DATA_BLOCK "ManualOperationControl_U1Em6"   // DB199
// stored: MemoryReserve 100
   VAR
      manualOperationEm { ExternalAccessible := 'False'; ExternalVisible := 'False'; ExternalWritable := 'False'} : "LAF_typeManEm";
      manualOperationEmArea { ExternalAccessible := 'False'; ExternalVisible := 'False'; ExternalWritable := 'False'} : Array[1..2] of "LAF_typeManOperationArea";
      manualOperationCms { ExternalAccessible := 'False'; ExternalVisible := 'False'; ExternalWritable := 'False'} : Array[1..90] of "LAF_typeManOperation";
      axis { ExternalAccessible := 'False'; ExternalVisible := 'False'; ExternalWritable := 'False'} : Array[0..0] of "LBC_typeAxisControlInterface";
      axis64Pos { S7_SetPoint := 'True'} : Array[0..20] of "LBC_typeAxis64PosInterface";
      softCam { S7_SetPoint := 'True'} : Array[0..20] of "LER_typeSoftCamInterface2";
      twoWayActuator { S7_SetPoint := 'True'} : Array[0..14] of "LBC_typeTwoWayActuatorInterface";
   END_VAR
BEGIN
   manualOperationEm.equipmentModuleNum := 1070;
   manualOperationEm.actvArea := 0;
   manualOperationEm.pages.total := 0;
   manualOperationEm.pages.actv := 0;
   manualOperationEm.pages.numOfActvItems := 0;
   manualOperationEmArea[1..2].areaNum := 0;
   manualOperationEmArea[1].displayedLines := '6-18;';
   manualOperationEmArea[2].displayedLines := '21-26;';
   manualOperationEmArea[1..2].hmiPage.total := 0;
   manualOperationEmArea[1..2].hmiPage.actv := 0;
   manualOperationEmArea[1..2].hmiPage.numOfActvItems := 0;
   manualOperationCms[1..90].intf.lineNum := 0;
   manualOperationCms[1..90].intf.mode := 1;
   manualOperationCms[1..90].intf.showLine := FALSE;
   manualOperationCms[1..90].intf.enableMechAddr := FALSE;
   manualOperationCms[1..90].intf.expandable := FALSE;
   manualOperationCms[1..90].intf.disableLineSel := FALSE;
   manualOperationCms[1..90].intf.enableBigArea := FALSE;
   manualOperationCms[1..90].intf.cnfrmExecLeft := FALSE;
   manualOperationCms[1..90].intf.cnfrmExecRight := FALSE;
   manualOperationCms[1..90].intf.disableLeft := FALSE;
   manualOperationCms[1..90].intf.disableRight := FALSE;
   manualOperationCms[1..90].intf.cnfrmExecLeftCmd := FALSE;
   manualOperationCms[1..90].intf.cnfrmExecRightCmd := FALSE;
   manualOperationCms[1..90].intf.fieldDevAckLeft := FALSE;
   manualOperationCms[1..90].intf.fieldDevAckRight := FALSE;
   manualOperationCms[1..90].intf.nextLeftEndPos := 0;
   manualOperationCms[1..90].intf.nextRightEndPos := 0;
   manualOperationCms[1].intf.leftEndPosSens[0..7] := FALSE;
   manualOperationCms[2].intf.leftEndPosSens[0..7] := FALSE;
   manualOperationCms[3].intf.leftEndPosSens[0..7] := FALSE;
   manualOperationCms[4].intf.leftEndPosSens[0..7] := FALSE;
   manualOperationCms[5].intf.leftEndPosSens[0..7] := FALSE;
   manualOperationCms[6].intf.leftEndPosSens[0..7] := FALSE;
   manualOperationCms[7].intf.leftEndPosSens[0..7] := FALSE;
   manualOperationCms[8].intf.leftEndPosSens[0..7] := FALSE;
   manualOperationCms[9].intf.leftEndPosSens[0..7] := FALSE;
   manualOperationCms[10].intf.leftEndPosSens[0..7] := FALSE;
   manualOperationCms[11].intf.leftEndPosSens[0..7] := FALSE;
   manualOperationCms[12].intf.leftEndPosSens[0..7] := FALSE;
   manualOperationCms[13].intf.leftEndPosSens[0..7] := FALSE;
   manualOperationCms[14].intf.leftEndPosSens[0..7] := FALSE;
   manualOperationCms[15].intf.leftEndPosSens[0..7] := FALSE;
   manualOperationCms[16].intf.leftEndPosSens[0..7] := FALSE;
   manualOperationCms[17].intf.leftEndPosSens[0..7] := FALSE;
   manualOperationCms[18].intf.leftEndPosSens[0..7] := FALSE;
   manualOperationCms[19].intf.leftEndPosSens[0..7] := FALSE;
   manualOperationCms[20].intf.leftEndPosSens[0..7] := FALSE;
   manualOperationCms[21].intf.leftEndPosSens[0..7] := FALSE;
   manualOperationCms[22].intf.leftEndPosSens[0..7] := FALSE;
   manualOperationCms[23].intf.leftEndPosSens[0..7] := FALSE;
   manualOperationCms[24].intf.leftEndPosSens[0..7] := FALSE;
   manualOperationCms[25].intf.leftEndPosSens[0..7] := FALSE;
   manualOperationCms[26].intf.leftEndPosSens[0..7] := FALSE;
   manualOperationCms[27].intf.leftEndPosSens[0..7] := FALSE;
   manualOperationCms[28].intf.leftEndPosSens[0..7] := FALSE;
   manualOperationCms[29].intf.leftEndPosSens[0..7] := FALSE;
   manualOperationCms[30].intf.leftEndPosSens[0..7] := FALSE;
   manualOperationCms[31].intf.leftEndPosSens[0..7] := FALSE;
   manualOperationCms[32].intf.leftEndPosSens[0..7] := FALSE;
   manualOperationCms[33].intf.leftEndPosSens[0..7] := FALSE;
   manualOperationCms[34].intf.leftEndPosSens[0..7] := FALSE;
   manualOperationCms[35].intf.leftEndPosSens[0..7] := FALSE;
   manualOperationCms[36].intf.leftEndPosSens[0..7] := FALSE;
   manualOperationCms[37].intf.leftEndPosSens[0..7] := FALSE;
   manualOperationCms[38].intf.leftEndPosSens[0..7] := FALSE;
   manualOperationCms[39].intf.leftEndPosSens[0..7] := FALSE;
   manualOperationCms[40].intf.leftEndPosSens[0..7] := FALSE;
   manualOperationCms[41].intf.leftEndPosSens[0..7] := FALSE;
   manualOperationCms[42].intf.leftEndPosSens[0..7] := FALSE;
   manualOperationCms[43].intf.leftEndPosSens[0..7] := FALSE;
   manualOperationCms[44].intf.leftEndPosSens[0..7] := FALSE;
   manualOperationCms[45].intf.leftEndPosSens[0..7] := FALSE;
   manualOperationCms[46].intf.leftEndPosSens[0..7] := FALSE;
   manualOperationCms[47].intf.leftEndPosSens[0..7] := FALSE;
   manualOperationCms[48].intf.leftEndPosSens[0..7] := FALSE;
   manualOperationCms[49].intf.leftEndPosSens[0..7] := FALSE;
   manualOperationCms[50].intf.leftEndPosSens[0..7] := FALSE;
   manualOperationCms[51].intf.leftEndPosSens[0..7] := FALSE;
   manualOperationCms[52].intf.leftEndPosSens[0..7] := FALSE;
   manualOperationCms[53].intf.leftEndPosSens[0..7] := FALSE;
   manualOperationCms[54].intf.leftEndPosSens[0..7] := FALSE;
   manualOperationCms[55].intf.leftEndPosSens[0..7] := FALSE;
   manualOperationCms[56].intf.leftEndPosSens[0..7] := FALSE;
   manualOperationCms[57].intf.leftEndPosSens[0..7] := FALSE;
   manualOperationCms[58].intf.leftEndPosSens[0..7] := FALSE;
   manualOperationCms[59].intf.leftEndPosSens[0..7] := FALSE;
   manualOperationCms[60].intf.leftEndPosSens[0..7] := FALSE;
   manualOperationCms[61].intf.leftEndPosSens[0..7] := FALSE;
   manualOperationCms[62].intf.leftEndPosSens[0..7] := FALSE;
   manualOperationCms[63].intf.leftEndPosSens[0..7] := FALSE;
   manualOperationCms[64].intf.leftEndPosSens[0..7] := FALSE;
   manualOperationCms[65].intf.leftEndPosSens[0..7] := FALSE;
   manualOperationCms[66].intf.leftEndPosSens[0..7] := FALSE;
   manualOperationCms[67].intf.leftEndPosSens[0..7] := FALSE;
   manualOperationCms[68].intf.leftEndPosSens[0..7] := FALSE;
   manualOperationCms[69].intf.leftEndPosSens[0..7] := FALSE;
   manualOperationCms[70].intf.leftEndPosSens[0..7] := FALSE;
   manualOperationCms[71].intf.leftEndPosSens[0..7] := FALSE;
   manualOperationCms[72].intf.leftEndPosSens[0..7] := FALSE;
   manualOperationCms[73].intf.leftEndPosSens[0..7] := FALSE;
   manualOperationCms[74].intf.leftEndPosSens[0..7] := FALSE;
   manualOperationCms[75].intf.leftEndPosSens[0..7] := FALSE;
   manualOperationCms[76].intf.leftEndPosSens[0..7] := FALSE;
   manualOperationCms[77].intf.leftEndPosSens[0..7] := FALSE;
   manualOperationCms[78].intf.leftEndPosSens[0..7] := FALSE;
   manualOperationCms[79].intf.leftEndPosSens[0..7] := FALSE;
   manualOperationCms[80].intf.leftEndPosSens[0..7] := FALSE;
   manualOperationCms[81].intf.leftEndPosSens[0..7] := FALSE;
   manualOperationCms[82].intf.leftEndPosSens[0..7] := FALSE;
   manualOperationCms[83].intf.leftEndPosSens[0..7] := FALSE;
   manualOperationCms[84].intf.leftEndPosSens[0..7] := FALSE;
   manualOperationCms[85].intf.leftEndPosSens[0..7] := FALSE;
   manualOperationCms[86].intf.leftEndPosSens[0..7] := FALSE;
   manualOperationCms[87].intf.leftEndPosSens[0..7] := FALSE;
   manualOperationCms[88].intf.leftEndPosSens[0..7] := FALSE;
   manualOperationCms[89].intf.leftEndPosSens[0..7] := FALSE;
   manualOperationCms[90].intf.leftEndPosSens[0..7] := FALSE;
   manualOperationCms[1].intf.rightEndPosSens[0..7] := FALSE;
   manualOperationCms[2].intf.rightEndPosSens[0..7] := FALSE;
   manualOperationCms[3].intf.rightEndPosSens[0..7] := FALSE;
   manualOperationCms[4].intf.rightEndPosSens[0..7] := FALSE;
   manualOperationCms[5].intf.rightEndPosSens[0..7] := FALSE;
   manualOperationCms[6].intf.rightEndPosSens[0..7] := FALSE;
   manualOperationCms[7].intf.rightEndPosSens[0..7] := FALSE;
   manualOperationCms[8].intf.rightEndPosSens[0..7] := FALSE;
   manualOperationCms[9].intf.rightEndPosSens[0..7] := FALSE;
   manualOperationCms[10].intf.rightEndPosSens[0..7] := FALSE;
   manualOperationCms[11].intf.rightEndPosSens[0..7] := FALSE;
   manualOperationCms[12].intf.rightEndPosSens[0..7] := FALSE;
   manualOperationCms[13].intf.rightEndPosSens[0..7] := FALSE;
   manualOperationCms[14].intf.rightEndPosSens[0..7] := FALSE;
   manualOperationCms[15].intf.rightEndPosSens[0..7] := FALSE;
   manualOperationCms[16].intf.rightEndPosSens[0..7] := FALSE;
   manualOperationCms[17].intf.rightEndPosSens[0..7] := FALSE;
   manualOperationCms[18].intf.rightEndPosSens[0..7] := FALSE;
   manualOperationCms[19].intf.rightEndPosSens[0..7] := FALSE;
   manualOperationCms[20].intf.rightEndPosSens[0..7] := FALSE;
   manualOperationCms[21].intf.rightEndPosSens[0..7] := FALSE;
   manualOperationCms[22].intf.rightEndPosSens[0..7] := FALSE;
   manualOperationCms[23].intf.rightEndPosSens[0..7] := FALSE;
   manualOperationCms[24].intf.rightEndPosSens[0..7] := FALSE;
   manualOperationCms[25].intf.rightEndPosSens[0..7] := FALSE;
   manualOperationCms[26].intf.rightEndPosSens[0..7] := FALSE;
   manualOperationCms[27].intf.rightEndPosSens[0..7] := FALSE;
   manualOperationCms[28].intf.rightEndPosSens[0..7] := FALSE;
   manualOperationCms[29].intf.rightEndPosSens[0..7] := FALSE;
   manualOperationCms[30].intf.rightEndPosSens[0..7] := FALSE;
   manualOperationCms[31].intf.rightEndPosSens[0..7] := FALSE;
   manualOperationCms[32].intf.rightEndPosSens[0..7] := FALSE;
   manualOperationCms[33].intf.rightEndPosSens[0..7] := FALSE;
   manualOperationCms[34].intf.rightEndPosSens[0..7] := FALSE;
   manualOperationCms[35].intf.rightEndPosSens[0..7] := FALSE;
   manualOperationCms[36].intf.rightEndPosSens[0..7] := FALSE;
   manualOperationCms[37].intf.rightEndPosSens[0..7] := FALSE;
   manualOperationCms[38].intf.rightEndPosSens[0..7] := FALSE;
   manualOperationCms[39].intf.rightEndPosSens[0..7] := FALSE;
   manualOperationCms[40].intf.rightEndPosSens[0..7] := FALSE;
   manualOperationCms[41].intf.rightEndPosSens[0..7] := FALSE;
   manualOperationCms[42].intf.rightEndPosSens[0..7] := FALSE;
   manualOperationCms[43].intf.rightEndPosSens[0..7] := FALSE;
   manualOperationCms[44].intf.rightEndPosSens[0..7] := FALSE;
   manualOperationCms[45].intf.rightEndPosSens[0..7] := FALSE;
   manualOperationCms[46].intf.rightEndPosSens[0..7] := FALSE;
   manualOperationCms[47].intf.rightEndPosSens[0..7] := FALSE;
   manualOperationCms[48].intf.rightEndPosSens[0..7] := FALSE;
   manualOperationCms[49].intf.rightEndPosSens[0..7] := FALSE;
   manualOperationCms[50].intf.rightEndPosSens[0..7] := FALSE;
   manualOperationCms[51].intf.rightEndPosSens[0..7] := FALSE;
   manualOperationCms[52].intf.rightEndPosSens[0..7] := FALSE;
   manualOperationCms[53].intf.rightEndPosSens[0..7] := FALSE;
   manualOperationCms[54].intf.rightEndPosSens[0..7] := FALSE;
   manualOperationCms[55].intf.rightEndPosSens[0..7] := FALSE;
   manualOperationCms[56].intf.rightEndPosSens[0..7] := FALSE;
   manualOperationCms[57].intf.rightEndPosSens[0..7] := FALSE;
   manualOperationCms[58].intf.rightEndPosSens[0..7] := FALSE;
   manualOperationCms[59].intf.rightEndPosSens[0..7] := FALSE;
   manualOperationCms[60].intf.rightEndPosSens[0..7] := FALSE;
   manualOperationCms[61].intf.rightEndPosSens[0..7] := FALSE;
   manualOperationCms[62].intf.rightEndPosSens[0..7] := FALSE;
   manualOperationCms[63].intf.rightEndPosSens[0..7] := FALSE;
   manualOperationCms[64].intf.rightEndPosSens[0..7] := FALSE;
   manualOperationCms[65].intf.rightEndPosSens[0..7] := FALSE;
   manualOperationCms[66].intf.rightEndPosSens[0..7] := FALSE;
   manualOperationCms[67].intf.rightEndPosSens[0..7] := FALSE;
   manualOperationCms[68].intf.rightEndPosSens[0..7] := FALSE;
   manualOperationCms[69].intf.rightEndPosSens[0..7] := FALSE;
   manualOperationCms[70].intf.rightEndPosSens[0..7] := FALSE;
   manualOperationCms[71].intf.rightEndPosSens[0..7] := FALSE;
   manualOperationCms[72].intf.rightEndPosSens[0..7] := FALSE;
   manualOperationCms[73].intf.rightEndPosSens[0..7] := FALSE;
   manualOperationCms[74].intf.rightEndPosSens[0..7] := FALSE;
   manualOperationCms[75].intf.rightEndPosSens[0..7] := FALSE;
   manualOperationCms[76].intf.rightEndPosSens[0..7] := FALSE;
   manualOperationCms[77].intf.rightEndPosSens[0..7] := FALSE;
   manualOperationCms[78].intf.rightEndPosSens[0..7] := FALSE;
   manualOperationCms[79].intf.rightEndPosSens[0..7] := FALSE;
   manualOperationCms[80].intf.rightEndPosSens[0..7] := FALSE;
   manualOperationCms[81].intf.rightEndPosSens[0..7] := FALSE;
   manualOperationCms[82].intf.rightEndPosSens[0..7] := FALSE;
   manualOperationCms[83].intf.rightEndPosSens[0..7] := FALSE;
   manualOperationCms[84].intf.rightEndPosSens[0..7] := FALSE;
   manualOperationCms[85].intf.rightEndPosSens[0..7] := FALSE;
   manualOperationCms[86].intf.rightEndPosSens[0..7] := FALSE;
   manualOperationCms[87].intf.rightEndPosSens[0..7] := FALSE;
   manualOperationCms[88].intf.rightEndPosSens[0..7] := FALSE;
   manualOperationCms[89].intf.rightEndPosSens[0..7] := FALSE;
   manualOperationCms[90].intf.rightEndPosSens[0..7] := FALSE;
   manualOperationCms[1..90].intf.pos := 0.0;
   manualOperationCms[1..90].intf.minPos := 0.0;
   manualOperationCms[1..90].intf.maxPos := 0.0;
   manualOperationCms[1..90].intf.showPos := 0;
   manualOperationCms[1..90].cmd.lineSel := FALSE;
   manualOperationCms[1..90].cmd.expandedOemArea := FALSE;
   manualOperationCms[1..90].cmd.execLeftCmd := FALSE;
   manualOperationCms[1..90].cmd.execRightCmd := FALSE;
   manualOperationCms[1..90].cmd.disableLeftClick := FALSE;
   manualOperationCms[1..90].cmd.disableRightClick := FALSE;
   manualOperationCms[1..90].cmd.moreInfo := FALSE;
   manualOperationCms[1..90].cmd.actvAddr := 1;
   axis[0].commandConfiguration.generalSettings.stopOnError := TRUE;
   axis[0].commandConfiguration.generalSettings.resetWithRestart := FALSE;
   axis[0].commandConfiguration.generalSettings.abortWaitingSyncCmd := TRUE;
   axis[0].commandConfiguration.power.startMode := 1;
   axis[0].commandConfiguration.power.stopMode := 0;
   axis[0].commandConfiguration.power.syncMotionSimulation := FALSE;
   axis[0].commandConfiguration.power.syncMotionSimulationExtendedMode := -1;
   axis[0].commandConfiguration.jog.velocity := 0.0;
   axis[0].commandConfiguration.jog.acceleration := -1.0;
   axis[0].commandConfiguration.jog.deceleration := -1.0;
   axis[0].commandConfiguration.jog.jerk := -1.0;
   axis[0].commandConfiguration.jog.positionControlled := TRUE;
   axis[0].commandConfiguration.jog.increment := 0.0;
   axis[0].commandConfiguration.jog.mode := 0;
   axis[0].commandConfiguration.moveVelocity.velocity := 0.0;
   axis[0].commandConfiguration.moveVelocity.acceleration := -1.0;
   axis[0].commandConfiguration.moveVelocity.deceleration := -1.0;
   axis[0].commandConfiguration.moveVelocity.jerk := -1.0;
   axis[0].commandConfiguration.moveVelocity.direction := 0;
   axis[0].commandConfiguration.moveVelocity.positionControlled := TRUE;
   axis[0].commandConfiguration.moveVelocity.velocityChangeOnTheFly := FALSE;
   axis[0].commandConfiguration.stop.deceleration := -1.0;
   axis[0].commandConfiguration.stop.jerk := -1.0;
   axis[0].commandConfiguration.stop.abortAcceleration := FALSE;
   axis[0].commandConfiguration.fastStop.deceleration := -1.0;
   axis[0].commandConfiguration.fastStop.jerk := -1.0;
   axis[0].commandConfiguration.fastStop.abortAcceleration := FALSE;
   axis[0].commandConfiguration.fastStop.replaceStopPossible := FALSE;
   axis[0].commandConfiguration.torqueLimiting.limit := -1.0;
   axis[0].commandConfiguration.torqueLimiting.mode := 0;
   axis[0].commandConfiguration.homing.position := 0.0;
   axis[0].commandConfiguration.homing.mode := 0;
   axis[0].commandConfiguration.homing.sensor := 0;
   axis[0].commandConfiguration.homing.extendedMode := -1;
   axis[0].commandConfiguration.homing.extendedModeTorqueLimit := 0.0;
   axis[0].commandConfiguration.homing.extendedModeTargetPosition := 0.0;
   axis[0].commandConfiguration.posRelative.distance := 0.0;
   axis[0].commandConfiguration.posRelative.velocity := -1.0;
   axis[0].commandConfiguration.posRelative.acceleration := -1.0;
   axis[0].commandConfiguration.posRelative.deceleration := -1.0;
   axis[0].commandConfiguration.posRelative.jerk := -1.0;
   axis[0].commandConfiguration.posRelative.direction := 0;
   axis[0].commandConfiguration.posAbsolute.position := 0.0;
   axis[0].commandConfiguration.posAbsolute.velocity := -1.0;
   axis[0].commandConfiguration.posAbsolute.acceleration := -1.0;
   axis[0].commandConfiguration.posAbsolute.deceleration := -1.0;
   axis[0].commandConfiguration.posAbsolute.jerk := -1.0;
   axis[0].commandConfiguration.posAbsolute.direction := 1;
   axis[0].commandConfiguration.posAbsolute.positionChangeOnTheFly := FALSE;
   axis[0].commandConfiguration.posAbsolute.velocityChangeOnTheFly := FALSE;
   axis[0].commandConfiguration.posSuperimposed.distance := 0.0;
   axis[0].commandConfiguration.posSuperimposed.velocityDiff := -1.0;
   axis[0].commandConfiguration.posSuperimposed.acceleration := -1.0;
   axis[0].commandConfiguration.posSuperimposed.deceleration := -1.0;
   axis[0].commandConfiguration.posSuperimposed.jerk := -1.0;
   axis[0].commandConfiguration.posSuperimposed.direction := 0;
   axis[0].commandConfiguration.haltSuperimposed.deceleration := -1.0;
   axis[0].commandConfiguration.haltSuperimposed.jerk := -1.0;
   axis[0].commandConfiguration.haltSuperimposed.abortAcceleration := FALSE;
   axis[0].commandConfiguration.gearInRelative.ratioNumerator := 1;
   axis[0].commandConfiguration.gearInRelative.ratioDenominator := 1;
   axis[0].commandConfiguration.gearInRelative.acceleration := -1.0;
   axis[0].commandConfiguration.gearInRelative.deceleration := -1.0;
   axis[0].commandConfiguration.gearInRelative.jerk := -1.0;
   axis[0].commandConfiguration.gearInRelative.ratioChangeOnTheFly := FALSE;
   axis[0].commandConfiguration.gearInAbsolute.ratioNumerator := 1;
   axis[0].commandConfiguration.gearInAbsolute.ratioDenominator := 1;
   axis[0].commandConfiguration.gearInAbsolute.masterSyncPosition := 0.0;
   axis[0].commandConfiguration.gearInAbsolute.slaveSyncPosition := 0.0;
   axis[0].commandConfiguration.gearInAbsolute.syncProfileReference := 1;
   axis[0].commandConfiguration.gearInAbsolute.masterStartDistance := 0.0;
   axis[0].commandConfiguration.gearInAbsolute.velocity := -1.0;
   axis[0].commandConfiguration.gearInAbsolute.acceleration := -1.0;
   axis[0].commandConfiguration.gearInAbsolute.deceleration := -1.0;
   axis[0].commandConfiguration.gearInAbsolute.jerk := -1.0;
   axis[0].commandConfiguration.gearInAbsolute.syncDirection := 1;
   axis[0].commandConfiguration.gearInAbsolute.ratioChangeOnTheFly := FALSE;
   axis[0].commandConfiguration.gearInVelocity.continuousUpdate := FALSE;
   axis[0].commandConfiguration.gearInVelocity.ratioNumerator := 1;
   axis[0].commandConfiguration.gearInVelocity.ratioDenominator := 1;
   axis[0].commandConfiguration.gearInVelocity.acceleration := -1.0;
   axis[0].commandConfiguration.gearInVelocity.deceleration := -1.0;
   axis[0].commandConfiguration.gearInVelocity.jerk := -1.0;
   axis[0].commandConfiguration.gearInVelocity.positionControlled := FALSE;
   axis[0].commandConfiguration.camIn.masterOffset := 0.0;
   axis[0].commandConfiguration.camIn.slaveOffset := 0.0;
   axis[0].commandConfiguration.camIn.masterScaling := 1.0;
   axis[0].commandConfiguration.camIn.slaveScaling := 1.0;
   axis[0].commandConfiguration.camIn.masterSyncPosition := 0.0;
   axis[0].commandConfiguration.camIn.syncProfileReference := 1;
   axis[0].commandConfiguration.camIn.masterStartDistance := 0.0;
   axis[0].commandConfiguration.camIn.velocity := -1.0;
   axis[0].commandConfiguration.camIn.acceleration := -1.0;
   axis[0].commandConfiguration.camIn.deceleration := -1.0;
   axis[0].commandConfiguration.camIn.jerk := -1.0;
   axis[0].commandConfiguration.camIn.applicationMode := 0;
   axis[0].commandConfiguration.camIn.syncDirection := 1;
   axis[0].commandConfiguration.gearOutCamOut.slavePosition := 0.0;
   axis[0].commandConfiguration.gearOutCamOut.syncProfileReference := 1;
   axis[0].commandConfiguration.gearOutCamOut.masterStopDistance := 0.0;
   axis[0].commandConfiguration.gearOutCamOut.deceleration := -1.0;
   axis[0].commandConfiguration.gearOutCamOut.jerk := -1.0;
   axis[0].commandConfiguration.gearOutCamOut.syncOutDirection := 3;
   axis[0].commandConfiguration.gearOutCamOut.gearOutCamOutMode := -1;
   axis[0].commandConfiguration.phasing.phaseShift := 0.0;
   axis[0].commandConfiguration.phasing.velocity := -1.0;
   axis[0].commandConfiguration.phasing.acceleration := -1.0;
   axis[0].commandConfiguration.phasing.deceleration := -1.0;
   axis[0].commandConfiguration.phasing.jerk := -1.0;
   axis[0].commandConfiguration.phasing.profileReference := 0;
   axis[0].commandConfiguration.phasing.phasingDistance := 0.0;
   axis[0].commandConfiguration.phasing.startPosition := 0.0;
   axis[0].commandConfiguration.phasing.direction := 3;
   axis[0].commandConfiguration.phasing.phaseAbsolute := TRUE;
   axis[0].commandConfiguration.phasing.phaseShiftChangeOnTheFly := FALSE;
   axis[0].commandConfiguration.offset.offset := 0.0;
   axis[0].commandConfiguration.offset.profileReference := 1;
   axis[0].commandConfiguration.offset.offsetDistance := 0.0;
   axis[0].commandConfiguration.offset.startPosition := 0.0;
   axis[0].commandConfiguration.offset.direction := 3;
   axis[0].commandConfiguration.offset.offsetAbsolute := TRUE;
   axis[0].commandConfiguration.offset.offsetChangeOnTheFly := FALSE;
   axis[0].commands.enable := FALSE;
   axis[0].commands.enableAxis := FALSE;
   axis[0].commands.resetAxis := FALSE;
   axis[0].commands.openBrake := FALSE;
   axis[0].commands.jogForward := FALSE;
   axis[0].commands.jogBackward := FALSE;
   axis[0].commands.moveVelocity := FALSE;
   axis[0].commands.stop := FALSE;
   axis[0].commands.fastStop := FALSE;
   axis[0].commands.torqueLimiting := FALSE;
   axis[0].commands.homing := FALSE;
   axis[0].commands.posRelative := FALSE;
   axis[0].commands.posAbsolute := FALSE;
   axis[0].commands.posSuperimposed := FALSE;
   axis[0].commands.haltSuperimposed := FALSE;
   axis[0].commands.gearInRelative := FALSE;
   axis[0].commands.gearInAbsolute := FALSE;
   axis[0].commands.gearInVelocity := FALSE;
   axis[0].commands.camIn := FALSE;
   axis[0].commands.gearOutCamOut := FALSE;
   axis[0].commands.phasing := FALSE;
   axis[0].commands.offset := FALSE;
   axis[0].commands.refreshConfiguration := FALSE;
   axis[0].commands.editConfiguration := FALSE;
   axis[0].commands.saveConfiguration := FALSE;
   axis[0].commands.uploadCurrentTorque := FALSE;
   axis[0].commands.reset := FALSE;
   axis[0].monitoring.enable := FALSE;
   axis[0].monitoring.referenceDesignator := WSTRING#'';
   axis[0].monitoring.enabled := FALSE;
   axis[0].monitoring.resetAxis := FALSE;
   axis[0].monitoring.moveVelocity := FALSE;
   axis[0].monitoring.fastStop := FALSE;
   axis[0].monitoring.stop := FALSE;
   axis[0].monitoring.homing := FALSE;
   axis[0].monitoring.posRelative := FALSE;
   axis[0].monitoring.posAbsolute := FALSE;
   axis[0].monitoring.posSuperimposed := FALSE;
   axis[0].monitoring.haltSuperimposed := FALSE;
   axis[0].monitoring.gearInRelative := FALSE;
   axis[0].monitoring.offset := FALSE;
   axis[0].monitoring.phasing := FALSE;
   axis[0].monitoring.gearOutCamOut := FALSE;
   axis[0].monitoring.camIn := FALSE;
   axis[0].monitoring.gearInVelocity := FALSE;
   axis[0].monitoring.gearInAbsolute := FALSE;
   axis[0].monitoring.reset := FALSE;
   axis[0].monitoring.enableAxis := FALSE;
   axis[0].monitoring.openBrake := FALSE;
   axis[0].monitoring.torqueLimiting := FALSE;
   axis[0].monitoring.enableManualCmds := FALSE;
   axis[0].monitoring.jogBackward := FALSE;
   axis[0].monitoring.jogForward := FALSE;
   axis[0].monitoring.brakeOpened := FALSE;
   axis[0].monitoring.axisEnabled := FALSE;
   axis[0].monitoring.resetActive := FALSE;
   axis[0].monitoring.inVelocity := FALSE;
   axis[0].monitoring.inLimitation := FALSE;
   axis[0].monitoring.inClamping := FALSE;
   axis[0].monitoring.startSync := FALSE;
   axis[0].monitoring.inSync := FALSE;
   axis[0].monitoring.inSimulation := FALSE;
   axis[0].monitoring.jogSelected := FALSE;
   axis[0].monitoring.moveVelocitySelected := FALSE;
   axis[0].monitoring.stopSelected := FALSE;
   axis[0].monitoring.fastStopSelected := FALSE;
   axis[0].monitoring.torqueLimitingSelected := FALSE;
   axis[0].monitoring.homingSelected := FALSE;
   axis[0].monitoring.posRelativeSelected := FALSE;
   axis[0].monitoring.posAbsoluteSelected := FALSE;
   axis[0].monitoring.posSuperimposedSelected := FALSE;
   axis[0].monitoring.haltSuperimposedSelected := FALSE;
   axis[0].monitoring.gearInRelativeSelected := FALSE;
   axis[0].monitoring.gearInAbsoluteSelected := FALSE;
   axis[0].monitoring.gearInVelocitySelected := FALSE;
   axis[0].monitoring.camInSelected := FALSE;
   axis[0].monitoring.gearOutCamOutSelected := FALSE;
   axis[0].monitoring.phasingSelected := FALSE;
   axis[0].monitoring.offsetSelected := FALSE;
   axis[0].monitoring.commandBusy := FALSE;
   axis[0].monitoring.commandDone := FALSE;
   axis[0].monitoring.commandAborted := FALSE;
   axis[0].monitoring.homingCommandBusy := FALSE;
   axis[0].monitoring.homingCommandDone := FALSE;
   axis[0].monitoring.homingCommandAborted := FALSE;
   axis[0].monitoring.superimposedBusy := FALSE;
   axis[0].monitoring.superimposedDone := FALSE;
   axis[0].monitoring.superimposedAborted := FALSE;
   axis[0].monitoring.interlockGeneral := FALSE;
   axis[0].monitoring.interlockJogForward := FALSE;
   axis[0].monitoring.interlockJogBackward := FALSE;
   axis[0].monitoring.interlockWarningGeneral := FALSE;
   axis[0].monitoring.interlockWarningJogForward := FALSE;
   axis[0].monitoring.interlockWarningJogBackward := FALSE;
   axis[0].monitoring.valid := FALSE;
   axis[0].monitoring.busy := FALSE;
   axis[0].monitoring.error := FALSE;
   axis[0].monitoring.status := 16#0000;
   axis[0].monitoring.subfunctionStatus := 16#0000;
   axis[0].monitoring.actualPosition := 0.0;
   axis[0].monitoring.actualSpeed := 0.0;
   axis[0].monitoring.speedUnit := 0;
   axis[0].monitoring.positionUnit := 0;
   axis[0].monitoring.axisStatus1 := 16#0000_0000;
   axis[0].monitoring.axisStatus2 := 16#0000_0000;
   axis[0].monitoring.axisType := 0;
   axis[0].monitoring.maxVelocity := 0.0;
   axis[0].monitoring.actualCurrent := 0.0;
   axis[0].monitoring.actualTorque := 0.0;
   axis[0].monitoring.velocityOverrideEnabled := FALSE;
   axis[0].monitoring.sinaParaError := FALSE;
   axis[0].monitoring.sinaParaStatus := 16#0000_0000;
   axis[0].configuration.referenceDesignator := WSTRING#'AxisControl';
   axis[0].configuration.disableAlarms := FALSE;
   axis[0].configuration.masterControlPopUp := TRUE;
   axis64Pos[0..13].commandConfiguration.generalSettings.stopOnError := TRUE;
   axis64Pos[0..13].commandConfiguration.generalSettings.resetWithRestart := FALSE;
   axis64Pos[0..13].commandConfiguration.generalSettings.abortWaitingSyncCmd := TRUE;
   axis64Pos[0..13].commandConfiguration.power.startMode := 1;
   axis64Pos[0..13].commandConfiguration.power.stopMode := 0;
   axis64Pos[0..13].commandConfiguration.power.syncMotionSimulation := FALSE;
   axis64Pos[0..13].commandConfiguration.power.syncMotionSimulationExtendedMode := -1;
   axis64Pos[0..13].commandConfiguration.jog.velocity := 0.0;
   axis64Pos[0..13].commandConfiguration.jog.acceleration := -1.0;
   axis64Pos[0..13].commandConfiguration.jog.deceleration := -1.0;
   axis64Pos[0..13].commandConfiguration.jog.jerk := -1.0;
   axis64Pos[0..13].commandConfiguration.jog.positionControlled := TRUE;
   axis64Pos[0..13].commandConfiguration.jog.increment := 0.0;
   axis64Pos[0..13].commandConfiguration.jog.mode := 0;
   axis64Pos[0..13].commandConfiguration.moveVelocity.velocity := 0.0;
   axis64Pos[0..13].commandConfiguration.moveVelocity.acceleration := -1.0;
   axis64Pos[0..13].commandConfiguration.moveVelocity.deceleration := -1.0;
   axis64Pos[0..13].commandConfiguration.moveVelocity.jerk := -1.0;
   axis64Pos[0..13].commandConfiguration.moveVelocity.direction := 0;
   axis64Pos[0..13].commandConfiguration.moveVelocity.positionControlled := TRUE;
   axis64Pos[0..13].commandConfiguration.moveVelocity.velocityChangeOnTheFly := FALSE;
   axis64Pos[0..13].commandConfiguration.stop.deceleration := -1.0;
   axis64Pos[0..13].commandConfiguration.stop.jerk := -1.0;
   axis64Pos[0..13].commandConfiguration.stop.abortAcceleration := FALSE;
   axis64Pos[0..13].commandConfiguration.fastStop.deceleration := -1.0;
   axis64Pos[0..13].commandConfiguration.fastStop.jerk := -1.0;
   axis64Pos[0..13].commandConfiguration.fastStop.abortAcceleration := FALSE;
   axis64Pos[0..13].commandConfiguration.fastStop.replaceStopPossible := FALSE;
   axis64Pos[0..13].commandConfiguration.torqueLimiting.limit := -1.0;
   axis64Pos[0..13].commandConfiguration.torqueLimiting.mode := 0;
   axis64Pos[0..13].commandConfiguration.homing.position := 0.0;
   axis64Pos[0..13].commandConfiguration.homing.mode := 0;
   axis64Pos[0..13].commandConfiguration.homing.sensor := 0;
   axis64Pos[0..13].commandConfiguration.homing.extendedMode := -1;
   axis64Pos[0..13].commandConfiguration.homing.extendedModeTorqueLimit := 0.0;
   axis64Pos[0..13].commandConfiguration.homing.extendedModeTargetPosition := 0.0;
   axis64Pos[0..13].commandConfiguration.posRelative.distance := 0.0;
   axis64Pos[0..13].commandConfiguration.posRelative.velocity := -1.0;
   axis64Pos[0..13].commandConfiguration.posRelative.acceleration := -1.0;
   axis64Pos[0..13].commandConfiguration.posRelative.deceleration := -1.0;
   axis64Pos[0..13].commandConfiguration.posRelative.jerk := -1.0;
   axis64Pos[0..13].commandConfiguration.posRelative.direction := 0;
   axis64Pos[0..13].commandConfiguration.posAbsolute.position := 0.0;
   axis64Pos[0..13].commandConfiguration.posAbsolute.velocity := -1.0;
   axis64Pos[0..13].commandConfiguration.posAbsolute.acceleration := -1.0;
   axis64Pos[0..13].commandConfiguration.posAbsolute.deceleration := -1.0;
   axis64Pos[0..13].commandConfiguration.posAbsolute.jerk := -1.0;
   axis64Pos[0..13].commandConfiguration.posAbsolute.direction := 1;
   axis64Pos[0..13].commandConfiguration.posAbsolute.positionChangeOnTheFly := FALSE;
   axis64Pos[0..13].commandConfiguration.posAbsolute.velocityChangeOnTheFly := FALSE;
   axis64Pos[0..13].commandConfiguration.posSuperimposed.distance := 0.0;
   axis64Pos[0..13].commandConfiguration.posSuperimposed.velocityDiff := -1.0;
   axis64Pos[0..13].commandConfiguration.posSuperimposed.acceleration := -1.0;
   axis64Pos[0..13].commandConfiguration.posSuperimposed.deceleration := -1.0;
   axis64Pos[0..13].commandConfiguration.posSuperimposed.jerk := -1.0;
   axis64Pos[0..13].commandConfiguration.posSuperimposed.direction := 0;
   axis64Pos[0..13].commandConfiguration.haltSuperimposed.deceleration := -1.0;
   axis64Pos[0..13].commandConfiguration.haltSuperimposed.jerk := -1.0;
   axis64Pos[0..13].commandConfiguration.haltSuperimposed.abortAcceleration := FALSE;
   axis64Pos[0..13].commandConfiguration.gearInRelative.ratioNumerator := 1;
   axis64Pos[0..13].commandConfiguration.gearInRelative.ratioDenominator := 1;
   axis64Pos[0..13].commandConfiguration.gearInRelative.acceleration := -1.0;
   axis64Pos[0..13].commandConfiguration.gearInRelative.deceleration := -1.0;
   axis64Pos[0..13].commandConfiguration.gearInRelative.jerk := -1.0;
   axis64Pos[0..13].commandConfiguration.gearInRelative.ratioChangeOnTheFly := FALSE;
   axis64Pos[0..13].commandConfiguration.gearInAbsolute.ratioNumerator := 1;
   axis64Pos[0..13].commandConfiguration.gearInAbsolute.ratioDenominator := 1;
   axis64Pos[0..13].commandConfiguration.gearInAbsolute.masterSyncPosition := 0.0;
   axis64Pos[0..13].commandConfiguration.gearInAbsolute.slaveSyncPosition := 0.0;
   axis64Pos[0..13].commandConfiguration.gearInAbsolute.syncProfileReference := 1;
   axis64Pos[0..13].commandConfiguration.gearInAbsolute.masterStartDistance := 0.0;
   axis64Pos[0..13].commandConfiguration.gearInAbsolute.velocity := -1.0;
   axis64Pos[0..13].commandConfiguration.gearInAbsolute.acceleration := -1.0;
   axis64Pos[0..13].commandConfiguration.gearInAbsolute.deceleration := -1.0;
   axis64Pos[0..13].commandConfiguration.gearInAbsolute.jerk := -1.0;
   axis64Pos[0..13].commandConfiguration.gearInAbsolute.syncDirection := 1;
   axis64Pos[0..13].commandConfiguration.gearInAbsolute.ratioChangeOnTheFly := FALSE;
   axis64Pos[0..13].commandConfiguration.gearInVelocity.continuousUpdate := FALSE;
   axis64Pos[0..13].commandConfiguration.gearInVelocity.ratioNumerator := 1;
   axis64Pos[0..13].commandConfiguration.gearInVelocity.ratioDenominator := 1;
   axis64Pos[0..13].commandConfiguration.gearInVelocity.acceleration := -1.0;
   axis64Pos[0..13].commandConfiguration.gearInVelocity.deceleration := -1.0;
   axis64Pos[0..13].commandConfiguration.gearInVelocity.jerk := -1.0;
   axis64Pos[0..13].commandConfiguration.gearInVelocity.positionControlled := FALSE;
   axis64Pos[0..13].commandConfiguration.camIn.masterOffset := 0.0;
   axis64Pos[0..13].commandConfiguration.camIn.slaveOffset := 0.0;
   axis64Pos[0..13].commandConfiguration.camIn.masterScaling := 1.0;
   axis64Pos[0..13].commandConfiguration.camIn.slaveScaling := 1.0;
   axis64Pos[0..13].commandConfiguration.camIn.masterSyncPosition := 0.0;
   axis64Pos[0..13].commandConfiguration.camIn.syncProfileReference := 1;
   axis64Pos[0..13].commandConfiguration.camIn.masterStartDistance := 0.0;
   axis64Pos[0..13].commandConfiguration.camIn.velocity := -1.0;
   axis64Pos[0..13].commandConfiguration.camIn.acceleration := -1.0;
   axis64Pos[0..13].commandConfiguration.camIn.deceleration := -1.0;
   axis64Pos[0..13].commandConfiguration.camIn.jerk := -1.0;
   axis64Pos[0..13].commandConfiguration.camIn.applicationMode := 0;
   axis64Pos[0..13].commandConfiguration.camIn.syncDirection := 1;
   axis64Pos[0..13].commandConfiguration.gearOutCamOut.slavePosition := 0.0;
   axis64Pos[0..13].commandConfiguration.gearOutCamOut.syncProfileReference := 1;
   axis64Pos[0..13].commandConfiguration.gearOutCamOut.masterStopDistance := 0.0;
   axis64Pos[0..13].commandConfiguration.gearOutCamOut.deceleration := -1.0;
   axis64Pos[0..13].commandConfiguration.gearOutCamOut.jerk := -1.0;
   axis64Pos[0..13].commandConfiguration.gearOutCamOut.syncOutDirection := 3;
   axis64Pos[0..13].commandConfiguration.gearOutCamOut.gearOutCamOutMode := -1;
   axis64Pos[0..13].commandConfiguration.phasing.phaseShift := 0.0;
   axis64Pos[0..13].commandConfiguration.phasing.velocity := -1.0;
   axis64Pos[0..13].commandConfiguration.phasing.acceleration := -1.0;
   axis64Pos[0..13].commandConfiguration.phasing.deceleration := -1.0;
   axis64Pos[0..13].commandConfiguration.phasing.jerk := -1.0;
   axis64Pos[0..13].commandConfiguration.phasing.profileReference := 0;
   axis64Pos[0..13].commandConfiguration.phasing.phasingDistance := 0.0;
   axis64Pos[0..13].commandConfiguration.phasing.startPosition := 0.0;
   axis64Pos[0..13].commandConfiguration.phasing.direction := 3;
   axis64Pos[0..13].commandConfiguration.phasing.phaseAbsolute := TRUE;
   axis64Pos[0..13].commandConfiguration.phasing.phaseShiftChangeOnTheFly := FALSE;
   axis64Pos[0..13].commandConfiguration.offset.offset := 0.0;
   axis64Pos[0..13].commandConfiguration.offset.profileReference := 1;
   axis64Pos[0..13].commandConfiguration.offset.offsetDistance := 0.0;
   axis64Pos[0..13].commandConfiguration.offset.startPosition := 0.0;
   axis64Pos[0..13].commandConfiguration.offset.direction := 3;
   axis64Pos[0..13].commandConfiguration.offset.offsetAbsolute := TRUE;
   axis64Pos[0..13].commandConfiguration.offset.offsetChangeOnTheFly := FALSE;
   axis64Pos[0..13].commands.enableMasterControl := FALSE;
   axis64Pos[0..13].commands.enableAxis := FALSE;
   axis64Pos[0..13].commands.resetAxis := FALSE;
   axis64Pos[0..13].commands.openBrake := FALSE;
   axis64Pos[0..13].commands.jogForward := FALSE;
   axis64Pos[0..13].commands.jogBackward := FALSE;
   axis64Pos[0..13].commands.moveVelocity := FALSE;
   axis64Pos[0..13].commands.stop := FALSE;
   axis64Pos[0..13].commands.fastStop := FALSE;
   axis64Pos[0..13].commands.torqueLimiting := FALSE;
   axis64Pos[0..13].commands.homing := FALSE;
   axis64Pos[0..13].commands.posRelative := FALSE;
   axis64Pos[0..13].commands.posAbsolute := FALSE;
   axis64Pos[0..13].commands.posSuperimposed := FALSE;
   axis64Pos[0..13].commands.haltSuperimposed := FALSE;
   axis64Pos[0..13].commands.selectSetPosition := 0;
   axis64Pos[0..13].commands.uploadParameters := FALSE;
   axis64Pos[0..13].commands.refreshConfiguration := FALSE;
   axis64Pos[0..13].commands.editConfiguration := FALSE;
   axis64Pos[0..13].commands.saveConfiguration := FALSE;
   axis64Pos[0..13].commands.uploadCurrentTorque := FALSE;
   axis64Pos[0..13].commands.reset := FALSE;
   axis64Pos[0..13].monitoring.enable := FALSE;
   axis64Pos[0..13].monitoring.referenceDesignator := WSTRING#'';
   axis64Pos[0..13].monitoring.enabled := FALSE;
   axis64Pos[0..13].monitoring.enableManualCmds := FALSE;
   axis64Pos[0..13].monitoring.reset := FALSE;
   axis64Pos[0..13].monitoring.resetAxis := FALSE;
   axis64Pos[0..13].monitoring.enableAxis := FALSE;
   axis64Pos[0..13].monitoring.openBrake := FALSE;
   axis64Pos[0..13].monitoring.jogBackward := FALSE;
   axis64Pos[0..13].monitoring.jogForward := FALSE;
   axis64Pos[0..13].monitoring.moveVelocity := FALSE;
   axis64Pos[0..13].monitoring.stop := FALSE;
   axis64Pos[0..13].monitoring.fastStop := FALSE;
   axis64Pos[0..13].monitoring.torqueLimiting := FALSE;
   axis64Pos[0..13].monitoring.homing := FALSE;
   axis64Pos[0..13].monitoring.posRelative := FALSE;
   axis64Pos[0..13].monitoring.posAbsolute := FALSE;
   axis64Pos[0..13].monitoring.posSuperimposed := FALSE;
   axis64Pos[0..13].monitoring.haltSuperimposed := FALSE;
   axis64Pos[0..13].monitoring.brakeOpened := FALSE;
   axis64Pos[0..13].monitoring.axisEnabled := FALSE;
   axis64Pos[0..13].monitoring.resetActive := FALSE;
   axis64Pos[0..13].monitoring.inVelocity := FALSE;
   axis64Pos[0..13].monitoring.inLimitation := FALSE;
   axis64Pos[0..13].monitoring.inClamping := FALSE;
   axis64Pos[0..13].monitoring.startSync := FALSE;
   axis64Pos[0..13].monitoring.inSync := FALSE;
   axis64Pos[0..13].monitoring.inSimulation := FALSE;
   axis64Pos[0..13].monitoring.jogSelected := FALSE;
   axis64Pos[0..13].monitoring.moveVelocitySelected := FALSE;
   axis64Pos[0..13].monitoring.stopSelected := FALSE;
   axis64Pos[0..13].monitoring.fastStopSelected := FALSE;
   axis64Pos[0..13].monitoring.torqueLimitingSelected := FALSE;
   axis64Pos[0..13].monitoring.homingSelected := FALSE;
   axis64Pos[0..13].monitoring.posRelativeSelected := FALSE;
   axis64Pos[0..13].monitoring.posAbsoluteSelected := FALSE;
   axis64Pos[0..13].monitoring.posSuperimposedSelected := FALSE;
   axis64Pos[0..13].monitoring.haltSuperimposedSelected := FALSE;
   axis64Pos[0..13].monitoring.commandBusy := FALSE;
   axis64Pos[0..13].monitoring.commandDone := FALSE;
   axis64Pos[0..13].monitoring.commandAborted := FALSE;
   axis64Pos[0..13].monitoring.homingCommandBusy := FALSE;
   axis64Pos[0..13].monitoring.homingCommandDone := FALSE;
   axis64Pos[0..13].monitoring.homingCommandAborted := FALSE;
   axis64Pos[0..13].monitoring.superimposedBusy := FALSE;
   axis64Pos[0..13].monitoring.superimposedDone := FALSE;
   axis64Pos[0..13].monitoring.superimposedAborted := FALSE;
   axis64Pos[0..13].monitoring.selectSetPosition := 0;
   axis64Pos[0..13].monitoring.selectionController := TRUE;
   axis64Pos[0..13].monitoring.interlockGeneral := FALSE;
   axis64Pos[0..13].monitoring.interlockJogForward := FALSE;
   axis64Pos[0..13].monitoring.interlockJogBackward := FALSE;
   axis64Pos[0..13].monitoring.interlockWarningGeneral := FALSE;
   axis64Pos[0..13].monitoring.interlockWarningJogForward := FALSE;
   axis64Pos[0..13].monitoring.interlockWarningJogBackward := FALSE;
   axis64Pos[0..13].monitoring.valid := FALSE;
   axis64Pos[0..13].monitoring.busy := FALSE;
   axis64Pos[0..13].monitoring.error := FALSE;
   axis64Pos[0..13].monitoring.status := 16#0000;
   axis64Pos[0..13].monitoring.subfunctionStatus := 16#0000;
   axis64Pos[0..13].monitoring.actualPosition := 0.0;
   axis64Pos[0..13].monitoring.actualSpeed := 0.0;
   axis64Pos[0..13].monitoring.speedUnit := 0;
   axis64Pos[0..13].monitoring.positionUnit := 0;
   axis64Pos[0..13].monitoring.axisType := 0;
   axis64Pos[0..13].monitoring.maxVelocity := 0.0;
   axis64Pos[0..13].monitoring.actualCurrent := 0.0;
   axis64Pos[0..13].monitoring.actualTorque := 0.0;
   axis64Pos[0..13].monitoring.velocityOverrideEnabled := FALSE;
   axis64Pos[0..13].monitoring.sinaParaError := FALSE;
   axis64Pos[0..13].monitoring.sinaParaStatus := 16#0000_0000;
   axis64Pos[0..13].configuration.referenceDesignator := WSTRING#'Axis64Pos';
   axis64Pos[0..13].configuration.disableAlarms := FALSE;
   axis64Pos[0..13].configuration.masterControlPopUp := TRUE;
   axis64Pos[0].configuration.setPositions[0..15].position := 0.0;
   axis64Pos[1].configuration.setPositions[0..15].position := 0.0;
   axis64Pos[2].configuration.setPositions[0..15].position := 0.0;
   axis64Pos[3].configuration.setPositions[0..15].position := 0.0;
   axis64Pos[4].configuration.setPositions[0..15].position := 0.0;
   axis64Pos[5].configuration.setPositions[0..15].position := 0.0;
   axis64Pos[6].configuration.setPositions[0..15].position := 0.0;
   axis64Pos[7].configuration.setPositions[0..15].position := 0.0;
   axis64Pos[8].configuration.setPositions[0..15].position := 0.0;
   axis64Pos[9].configuration.setPositions[0..15].position := 0.0;
   axis64Pos[10].configuration.setPositions[0..15].position := 0.0;
   axis64Pos[11].configuration.setPositions[0..15].position := 0.0;
   axis64Pos[12].configuration.setPositions[0..15].position := 0.0;
   axis64Pos[13].configuration.setPositions[0..15].position := 0.0;
   axis64Pos[0].configuration.setPositions[0..15].velocity := -1.0;
   axis64Pos[1].configuration.setPositions[0..15].velocity := -1.0;
   axis64Pos[2].configuration.setPositions[0..15].velocity := -1.0;
   axis64Pos[3].configuration.setPositions[0..15].velocity := -1.0;
   axis64Pos[4].configuration.setPositions[0..15].velocity := -1.0;
   axis64Pos[5].configuration.setPositions[0..15].velocity := -1.0;
   axis64Pos[6].configuration.setPositions[0..15].velocity := -1.0;
   axis64Pos[7].configuration.setPositions[0..15].velocity := -1.0;
   axis64Pos[8].configuration.setPositions[0..15].velocity := -1.0;
   axis64Pos[9].configuration.setPositions[0..15].velocity := -1.0;
   axis64Pos[10].configuration.setPositions[0..15].velocity := -1.0;
   axis64Pos[11].configuration.setPositions[0..15].velocity := -1.0;
   axis64Pos[12].configuration.setPositions[0..15].velocity := -1.0;
   axis64Pos[13].configuration.setPositions[0..15].velocity := -1.0;
   axis64Pos[0].configuration.setPositions[0..15].acceleration := -1.0;
   axis64Pos[1].configuration.setPositions[0..15].acceleration := -1.0;
   axis64Pos[2].configuration.setPositions[0..15].acceleration := -1.0;
   axis64Pos[3].configuration.setPositions[0..15].acceleration := -1.0;
   axis64Pos[4].configuration.setPositions[0..15].acceleration := -1.0;
   axis64Pos[5].configuration.setPositions[0..15].acceleration := -1.0;
   axis64Pos[6].configuration.setPositions[0..15].acceleration := -1.0;
   axis64Pos[7].configuration.setPositions[0..15].acceleration := -1.0;
   axis64Pos[8].configuration.setPositions[0..15].acceleration := -1.0;
   axis64Pos[9].configuration.setPositions[0..15].acceleration := -1.0;
   axis64Pos[10].configuration.setPositions[0..15].acceleration := -1.0;
   axis64Pos[11].configuration.setPositions[0..15].acceleration := -1.0;
   axis64Pos[12].configuration.setPositions[0..15].acceleration := -1.0;
   axis64Pos[13].configuration.setPositions[0..15].acceleration := -1.0;
   axis64Pos[0].configuration.setPositions[0..15].deceleration := -1.0;
   axis64Pos[1].configuration.setPositions[0..15].deceleration := -1.0;
   axis64Pos[2].configuration.setPositions[0..15].deceleration := -1.0;
   axis64Pos[3].configuration.setPositions[0..15].deceleration := -1.0;
   axis64Pos[4].configuration.setPositions[0..15].deceleration := -1.0;
   axis64Pos[5].configuration.setPositions[0..15].deceleration := -1.0;
   axis64Pos[6].configuration.setPositions[0..15].deceleration := -1.0;
   axis64Pos[7].configuration.setPositions[0..15].deceleration := -1.0;
   axis64Pos[8].configuration.setPositions[0..15].deceleration := -1.0;
   axis64Pos[9].configuration.setPositions[0..15].deceleration := -1.0;
   axis64Pos[10].configuration.setPositions[0..15].deceleration := -1.0;
   axis64Pos[11].configuration.setPositions[0..15].deceleration := -1.0;
   axis64Pos[12].configuration.setPositions[0..15].deceleration := -1.0;
   axis64Pos[13].configuration.setPositions[0..15].deceleration := -1.0;
   axis64Pos[0].configuration.setPositions[0..15]."name" := '';
   axis64Pos[1].configuration.setPositions[0..15]."name" := '';
   axis64Pos[2].configuration.setPositions[0..15]."name" := '';
   axis64Pos[3].configuration.setPositions[0..15]."name" := '';
   axis64Pos[4].configuration.setPositions[0..15]."name" := '';
   axis64Pos[5].configuration.setPositions[0..15]."name" := '';
   axis64Pos[6].configuration.setPositions[0..15]."name" := '';
   axis64Pos[7].configuration.setPositions[0..15]."name" := '';
   axis64Pos[8].configuration.setPositions[0..15]."name" := '';
   axis64Pos[9].configuration.setPositions[0..15]."name" := '';
   axis64Pos[10].configuration.setPositions[0..15]."name" := '';
   axis64Pos[11].configuration.setPositions[0..15]."name" := '';
   axis64Pos[12].configuration.setPositions[0..15]."name" := '';
   axis64Pos[13].configuration.setPositions[0..15]."name" := '';
   twoWayActuator[0..6].commands.refreshConfiguration := FALSE;
   twoWayActuator[0..6].commands.editConfiguration := FALSE;
   twoWayActuator[0..6].commands.saveConfiguration := FALSE;
   twoWayActuator[0..6].commands.reset := FALSE;
   twoWayActuator[0..6].commands.commandHomePos := FALSE;
   twoWayActuator[0..6].commands.commandWorkPos := FALSE;
   twoWayActuator[0..6].monitoring.enable := FALSE;
   twoWayActuator[0..6].monitoring.referenceDesignator := WSTRING#'';
   twoWayActuator[0..6].monitoring.commandHomePos := FALSE;
   twoWayActuator[0..6].monitoring.commandWorkPos := FALSE;
   twoWayActuator[0..6].monitoring.goToHomePos := FALSE;
   twoWayActuator[0..6].monitoring.goToWorkPos := FALSE;
   twoWayActuator[0..6].monitoring.inHomePos := FALSE;
   twoWayActuator[0..6].monitoring.inWorkPos := FALSE;
   twoWayActuator[0..6].monitoring.reset := FALSE;
   twoWayActuator[0..6].monitoring.enableManualCmds := FALSE;
   twoWayActuator[0..6].monitoring.error := FALSE;
   twoWayActuator[0..6].monitoring.interlockHomePos := FALSE;
   twoWayActuator[0..6].monitoring.interlockWorkPos := FALSE;
   twoWayActuator[0..6].monitoring.status := 16#0000;
   twoWayActuator[0..6].monitoring.interlockWarningWorkPos := FALSE;
   twoWayActuator[0..6].monitoring.interlockWarningHomePos := FALSE;
   twoWayActuator[0..6].configuration.referenceDesignator := WSTRING#'TwoWayAct.';
   twoWayActuator[0..6].configuration.monitoringLeavingFeedback := T#5S;
   twoWayActuator[0..6].configuration.monitoringReachingFeedback := T#5S;
   twoWayActuator[0..6].configuration.monitoringDiscrepancy := T#0MS;
   twoWayActuator[0..6].configuration.setOutputHomeContinuously := TRUE;
   twoWayActuator[0..6].configuration.setOutputWorkContinuously := TRUE;
   twoWayActuator[0..6].configuration.disableHomeCommand := FALSE;
   twoWayActuator[0..6].configuration.disableFeedbackHomePos := FALSE;
   twoWayActuator[0..6].configuration.disableFeedbackWorkPos := FALSE;
   twoWayActuator[0..6].configuration.disableAlarms := FALSE;
   twoWayActuator[0..6].configuration.resetOutputsOnError := FALSE;
   twoWayActuator[0..6].configuration.allwaysWaitOnReachingTime := FALSE;
END_DATA_BLOCK

DATA_BLOCK "ManualOperationControl_U1Em7"   // DB201
// stored: MemoryReserve 100
   VAR
      manualOperationEm { ExternalAccessible := 'False'; ExternalVisible := 'False'; ExternalWritable := 'False'} : "LAF_typeManEm";
      manualOperationEmArea { ExternalAccessible := 'False'; ExternalVisible := 'False'; ExternalWritable := 'False'} : Array[1..2] of "LAF_typeManOperationArea";
      manualOperationCms { ExternalAccessible := 'False'; ExternalVisible := 'False'; ExternalWritable := 'False'} : Array[1..90] of "LAF_typeManOperation";
      axis { ExternalAccessible := 'False'; ExternalVisible := 'False'; ExternalWritable := 'False'} : Array[0..0] of "LBC_typeAxisControlInterface";
      axis64Pos { S7_SetPoint := 'True'} : Array[0..20] of "LBC_typeAxis64PosInterface";
      softCam { S7_SetPoint := 'True'} : Array[0..20] of "LER_typeSoftCamInterface2";
      twoWayActuator { S7_SetPoint := 'True'} : Array[0..14] of "LBC_typeTwoWayActuatorInterface";
   END_VAR
BEGIN
END_DATA_BLOCK

DATA_BLOCK "DriveDiagConfig"   // DB18
TITLE = DriveDiagConfig
AUTHOR : Siemens Digital Industries
FAMILY : LAF
NAME : LAF_DriveDiagConfigData
VERSION : 1.1
// Configuration data array for drive diagnostic
// stored: MemoryReserve 100
   VAR
      driveObjects : Array[0..41] of "LAF_typeDriveDiagConfig";
   END_VAR
BEGIN
   driveObjects[0].referenceDesignator := WSTRING#'BA030AZSDR1';
   driveObjects[1].referenceDesignator := WSTRING#'BA030AZSDR2';
   driveObjects[2].referenceDesignator := WSTRING#'BA030AZSDR3';
   driveObjects[3].referenceDesignator := WSTRING#'';
   driveObjects[4].referenceDesignator := WSTRING#'BA030AZSDR5';
   driveObjects[5].referenceDesignator := WSTRING#'BA030AZSDR6';
   driveObjects[6].referenceDesignator := WSTRING#'BA030AZSDR7';
   driveObjects[7].referenceDesignator := WSTRING#'BA030AZSDR8';
   driveObjects[8].referenceDesignator := WSTRING#'BA030AZSDR9';
   driveObjects[9].referenceDesignator := WSTRING#'BA030AZSDR10';
   driveObjects[10].referenceDesignator := WSTRING#'BA030AZSDR11';
   driveObjects[11].referenceDesignator := WSTRING#'BA030AZSDR12';
   driveObjects[12].referenceDesignator := WSTRING#'BA030AZSDR13';
   driveObjects[13].referenceDesignator := WSTRING#'BA030AZSDR14';
   driveObjects[14].referenceDesignator := WSTRING#'BA030AZSDR15';
   driveObjects[15].referenceDesignator := WSTRING#'BA030AZSDR16';
   driveObjects[16].referenceDesignator := WSTRING#'BA030AZSDR17';
   driveObjects[17].referenceDesignator := WSTRING#'BA030AZSDR18';
   driveObjects[18].referenceDesignator := WSTRING#'BA030AZSDR19';
   driveObjects[19].referenceDesignator := WSTRING#'BA030AZSDR20';
   driveObjects[20].referenceDesignator := WSTRING#'BA030AZSDR21';
   driveObjects[21].referenceDesignator := WSTRING#'BA030AZSDR22';
   driveObjects[22].referenceDesignator := WSTRING#'BA030AZSDR23';
   driveObjects[23].referenceDesignator := WSTRING#'BA030AZSDR24';
   driveObjects[24].referenceDesignator := WSTRING#'BA030AZSDR25';
   driveObjects[25].referenceDesignator := WSTRING#'BA030AZSDR26';
   driveObjects[26].referenceDesignator := WSTRING#'BA030AZSDR27';
   driveObjects[27].referenceDesignator := WSTRING#'BA030AZSDR28';
   driveObjects[28].referenceDesignator := WSTRING#'BA030AZSDR29';
   driveObjects[29].referenceDesignator := WSTRING#'BA030AZSDR30';
   driveObjects[30].referenceDesignator := WSTRING#'BA030AZSDR31';
   driveObjects[31].referenceDesignator := WSTRING#'BA030AZSDR32';
   driveObjects[32].referenceDesignator := WSTRING#'BA030AZSDR33';
   driveObjects[33].referenceDesignator := WSTRING#'BA030AZSDR34';
   driveObjects[34].referenceDesignator := WSTRING#'BA030AZSDR35';
   driveObjects[35].referenceDesignator := WSTRING#'BA030AZSDR36';
   driveObjects[36].referenceDesignator := WSTRING#'BA030AZSDR37';
   driveObjects[37].referenceDesignator := WSTRING#'BA030AZSDR38';
   driveObjects[38].referenceDesignator := WSTRING#'BA030AZSDR39';
   driveObjects[39].referenceDesignator := WSTRING#'BA030AZSDR40';
   driveObjects[40].referenceDesignator := WSTRING#'BA030AZSDR41';
   driveObjects[41].referenceDesignator := WSTRING#'';
   driveObjects[0].axisDB := 263;
   driveObjects[1].axisDB := 141;
   driveObjects[2].axisDB := 143;
   driveObjects[3].axisDB := 0;
   driveObjects[4].axisDB := 144;
   driveObjects[5].axisDB := 145;
   driveObjects[6].axisDB := 146;
   driveObjects[7].axisDB := 147;
   driveObjects[8].axisDB := 152;
   driveObjects[9].axisDB := 151;
   driveObjects[10].axisDB := 148;
   driveObjects[11].axisDB := 149;
   driveObjects[12].axisDB := 153;
   driveObjects[13].axisDB := 150;
   driveObjects[14].axisDB := 154;
   driveObjects[15].axisDB := 155;
   driveObjects[16].axisDB := 156;
   driveObjects[17].axisDB := 157;
   driveObjects[18].axisDB := 158;
   driveObjects[19].axisDB := 159;
   driveObjects[20].axisDB := 171;
   driveObjects[21].axisDB := 172;
   driveObjects[22].axisDB := 163;
   driveObjects[23].axisDB := 162;
   driveObjects[24].axisDB := 167;
   driveObjects[25].axisDB := 166;
   driveObjects[26].axisDB := 161;
   driveObjects[27].axisDB := 160;
   driveObjects[28].axisDB := 165;
   driveObjects[29].axisDB := 164;
   driveObjects[30].axisDB := 168;
   driveObjects[31].axisDB := 169;
   driveObjects[32].axisDB := 170;
   driveObjects[33].axisDB := 177;
   driveObjects[34].axisDB := 175;
   driveObjects[35].axisDB := 178;
   driveObjects[36].axisDB := 173;
   driveObjects[37].axisDB := 174;
   driveObjects[38].axisDB := 180;
   driveObjects[39].axisDB := 179;
   driveObjects[40].axisDB := 176;
   driveObjects[41].axisDB := 0;
   driveObjects[0..2].sinaType := 124;
   driveObjects[3].sinaType := 0;
   driveObjects[4..40].sinaType := 124;
   driveObjects[41].sinaType := 0;
   driveObjects[0].sinaHwID := 259;
   driveObjects[1].sinaHwID := 517;
   driveObjects[2].sinaHwID := 818;
   driveObjects[3].sinaHwID := 0;
   driveObjects[4].sinaHwID := 519;
   driveObjects[5].sinaHwID := 523;
   driveObjects[6].sinaHwID := 527;
   driveObjects[7].sinaHwID := 529;
   driveObjects[8].sinaHwID := 541;
   driveObjects[9].sinaHwID := 547;
   driveObjects[10].sinaHwID := 559;
   driveObjects[11].sinaHwID := 561;
   driveObjects[12].sinaHwID := 564;
   driveObjects[13].sinaHwID := 569;
   driveObjects[14].sinaHwID := 568;
   driveObjects[15].sinaHwID := 571;
   driveObjects[16].sinaHwID := 573;
   driveObjects[17].sinaHwID := 577;
   driveObjects[18].sinaHwID := 659;
   driveObjects[19].sinaHwID := 660;
   driveObjects[20].sinaHwID := 589;
   driveObjects[21].sinaHwID := 596;
   driveObjects[22].sinaHwID := 654;
   driveObjects[23].sinaHwID := 667;
   driveObjects[24].sinaHwID := 671;
   driveObjects[25].sinaHwID := 682;
   driveObjects[26].sinaHwID := 620;
   driveObjects[27].sinaHwID := 626;
   driveObjects[28].sinaHwID := 684;
   driveObjects[29].sinaHwID := 686;
   driveObjects[30].sinaHwID := 605;
   driveObjects[31].sinaHwID := 635;
   driveObjects[32].sinaHwID := 663;
   driveObjects[33].sinaHwID := 690;
   driveObjects[34].sinaHwID := 649;
   driveObjects[35].sinaHwID := 692;
   driveObjects[36].sinaHwID := 657;
   driveObjects[37].sinaHwID := 697;
   driveObjects[38].sinaHwID := 665;
   driveObjects[39].sinaHwID := 666;
   driveObjects[40].sinaHwID := 653;
   driveObjects[41].sinaHwID := 0;
   driveObjects[0..1].sinaDriveObjectNo := 3;
   driveObjects[2].sinaDriveObjectNo := 4;
   driveObjects[3].sinaDriveObjectNo := 1;
   driveObjects[4].sinaDriveObjectNo := 2;
   driveObjects[5].sinaDriveObjectNo := 3;
   driveObjects[6].sinaDriveObjectNo := 4;
   driveObjects[7].sinaDriveObjectNo := 10;
   driveObjects[8].sinaDriveObjectNo := 5;
   driveObjects[9..10].sinaDriveObjectNo := 6;
   driveObjects[11].sinaDriveObjectNo := 2;
   driveObjects[12].sinaDriveObjectNo := 3;
   driveObjects[13].sinaDriveObjectNo := 4;
   driveObjects[14..40].sinaDriveObjectNo := 5;
   driveObjects[41].sinaDriveObjectNo := 1;
END_DATA_BLOCK

DATA_BLOCK "DriveDiagInterfaceHmi"   // DB46
TITLE = DriveDiagInterfaceHmi
AUTHOR : Siemens Digital Industries
FAMILY : LAF
NAME : LAF_DriveDiagInterfaceHmi
VERSION : 1.1
// HMI interface for drive diagnostic
// stored: MemoryReserve 100
   VAR
      diagStatus : "LAF_typeDriveDiagInterfaceHmi";
   END_VAR
BEGIN
   diagStatus.hmi.referenceDesignator := WSTRING#'';
   diagStatus.hmi.driveIndex := 0;
   diagStatus.hmi.axisStatusScreenActive := FALSE;
   diagStatus.hmi.sinaStatusScreenActive := FALSE;
   diagStatus.hmi.sinaAlarmScreenActive := FALSE;
   diagStatus.hmi.sinaEposScreenActive := FALSE;
   diagStatus.hmi.sinaSafetyScreenActive := FALSE;
   diagStatus.axis."type" := 0;
   diagStatus.axis.values.position := 0.0;
   diagStatus.axis.values.velocity := 0.0;
   diagStatus.axis.values.actualPosition := 0.0;
   diagStatus.axis.values.actualVelocity := 0.0;
   diagStatus.axis.values.actualSpeed := 0.0;
   diagStatus.axis.statusAxis.statusWord := 16#0000_0000;
   diagStatus.axis.statusAxis.statusWord2 := 16#0000_0000;
   diagStatus.axis.statusAxis.warningWord := 16#0000_0000;
   diagStatus.axis.statusAxis.errorWord := 16#0000_0000;
   diagStatus.axis.statusAxis.status.bit00_Enable := FALSE;
   diagStatus.axis.statusAxis.status.bit01_Error := FALSE;
   diagStatus.axis.statusAxis.status.bit02_RestartActive := FALSE;
   diagStatus.axis.statusAxis.status.bit03_OnlineStartValuesChanged := FALSE;
   diagStatus.axis.statusAxis.status.bit04_ControlPanelActive := FALSE;
   diagStatus.axis.statusAxis.status.bit05_HomingDone := FALSE;
   diagStatus.axis.statusAxis.status.bit06_Done := FALSE;
   diagStatus.axis.statusAxis.status.bit07_Standstill := FALSE;
   diagStatus.axis.statusAxis.status.bit08_PositioningCommand := FALSE;
   diagStatus.axis.statusAxis.status.bit09_JogCommand := FALSE;
   diagStatus.axis.statusAxis.status.bit10_VelocityCommand := FALSE;
   diagStatus.axis.statusAxis.status.bit11_HomingCommand := FALSE;
   diagStatus.axis.statusAxis.status.bit12_ConstantVelocity := FALSE;
   diagStatus.axis.statusAxis.status.bit13_Accelerating := FALSE;
   diagStatus.axis.statusAxis.status.bit14_Decelerating := FALSE;
   diagStatus.axis.statusAxis.status.bit15_SWLimitMinActive := FALSE;
   diagStatus.axis.statusAxis.status.bit16_SWLimitMaxActive := FALSE;
   diagStatus.axis.statusAxis.status.bit17_HWLimitMinActive := FALSE;
   diagStatus.axis.statusAxis.status.bit18_HWLimitMaxActive := FALSE;
   diagStatus.axis.statusAxis.status.bit19_Reserved := FALSE;
   diagStatus.axis.statusAxis.status.bit20_Reserved := FALSE;
   diagStatus.axis.statusAxis.status.bit21_Synchronizing := FALSE;
   diagStatus.axis.statusAxis.status.bit22_Synchronous := FALSE;
   diagStatus.axis.statusAxis.status.bit23_SuperimposedMotionCommand := FALSE;
   diagStatus.axis.statusAxis.status.bit24_PhasingCommand := FALSE;
   diagStatus.axis.statusAxis.status.bit25_AxisSimulation := FALSE;
   diagStatus.axis.statusAxis.status.bit26_TorqueLimitingCommand := FALSE;
   diagStatus.axis.statusAxis.status.bit27_InLimitation := FALSE;
   diagStatus.axis.statusAxis.status.bit28_NonPositionControlled := FALSE;
   diagStatus.axis.statusAxis.status.bit29_KinematicsMotionCommand := FALSE;
   diagStatus.axis.statusAxis.status.bit30_InClamping := FALSE;
   diagStatus.axis.statusAxis.status.bit31_MotionInCommand := FALSE;
   diagStatus.axis.statusAxis.status2.bit00_StopCommand := FALSE;
   diagStatus.axis.statusAxis.status2.bit01_DesynchronizingCommand := FALSE;
   diagStatus.axis.statusAxis.status2.bit02_PassingBacklash := FALSE;
   diagStatus.axis.statusAxis.status2.bit03_PhasingCommandWaiting := FALSE;
   diagStatus.axis.statusAxis.status2.bit04_OffsetCommand := FALSE;
   diagStatus.axis.statusAxis.status2.bit05_OffsetCommandWaiting := FALSE;
   diagStatus.axis.statusAxis.status2.bit06_MotionInSuperimposedCommand := FALSE;
   diagStatus.axis.statusAxis.status2.bit07_HaltSuperimposedCommand := FALSE;
   diagStatus.axis.statusAxis.status2.bit08_Reserved := FALSE;
   diagStatus.axis.statusAxis.status2.bit09_Reserved := FALSE;
   diagStatus.axis.statusAxis.status2.bit10_Reserved := FALSE;
   diagStatus.axis.statusAxis.status2.bit11_Reserved := FALSE;
   diagStatus.axis.statusAxis.status2.bit12_Reserved := FALSE;
   diagStatus.axis.statusAxis.status2.bit13_Reserved := FALSE;
   diagStatus.axis.statusAxis.status2.bit14_Reserved := FALSE;
   diagStatus.axis.statusAxis.status2.bit15_Reserved := FALSE;
   diagStatus.axis.statusAxis.status2.bit16_Reserved := FALSE;
   diagStatus.axis.statusAxis.status2.bit17_Reserved := FALSE;
   diagStatus.axis.statusAxis.status2.bit18_Reserved := FALSE;
   diagStatus.axis.statusAxis.status2.bit19_Reserved := FALSE;
   diagStatus.axis.statusAxis.status2.bit20_Reserved := FALSE;
   diagStatus.axis.statusAxis.status2.bit21_Reserved := FALSE;
   diagStatus.axis.statusAxis.status2.bit22_Reserved := FALSE;
   diagStatus.axis.statusAxis.status2.bit23_Reserved := FALSE;
   diagStatus.axis.statusAxis.status2.bit24_Reserved := FALSE;
   diagStatus.axis.statusAxis.status2.bit25_Reserved := FALSE;
   diagStatus.axis.statusAxis.status2.bit26_Reserved := FALSE;
   diagStatus.axis.statusAxis.status2.bit27_Reserved := FALSE;
   diagStatus.axis.statusAxis.status2.bit28_Reserved := FALSE;
   diagStatus.axis.statusAxis.status2.bit29_Reserved := FALSE;
   diagStatus.axis.statusAxis.status2.bit30_Reserved := FALSE;
   diagStatus.axis.statusAxis.status2.bit31_Reserved := FALSE;
   diagStatus.axis.statusAxis.warning.bit00_SystemWarning := FALSE;
   diagStatus.axis.statusAxis.warning.bit01_ConfigWarning := FALSE;
   diagStatus.axis.statusAxis.warning.bit02_UserWarning := FALSE;
   diagStatus.axis.statusAxis.warning.bit03_CommandNotAccepted := FALSE;
   diagStatus.axis.statusAxis.warning.bit04_DriveWarning := FALSE;
   diagStatus.axis.statusAxis.warning.bit05_SensorWarning := FALSE;
   diagStatus.axis.statusAxis.warning.bit06_DynamicWarning := FALSE;
   diagStatus.axis.statusAxis.warning.bit07_CommunicationWarning := FALSE;
   diagStatus.axis.statusAxis.warning.bit08_SWLimitMin := FALSE;
   diagStatus.axis.statusAxis.warning.bit09_SWLimitMax := FALSE;
   diagStatus.axis.statusAxis.warning.bit10_HomingWarning := FALSE;
   diagStatus.axis.statusAxis.warning.bit11_FollowingErrorWarning := FALSE;
   diagStatus.axis.statusAxis.warning.bit12_PositioningWarning := FALSE;
   diagStatus.axis.statusAxis.warning.bit13_PeripheralWarning := FALSE;
   diagStatus.axis.statusAxis.warning.bit14_SynchronousWarning := FALSE;
   diagStatus.axis.statusAxis.warning.bit15_AdaptionWarning := FALSE;
   diagStatus.axis.statusAxis.warning.bit16_Reserved := FALSE;
   diagStatus.axis.statusAxis.warning.bit17_Reserved := FALSE;
   diagStatus.axis.statusAxis.warning.bit18_Reserved := FALSE;
   diagStatus.axis.statusAxis.warning.bit19_Reserved := FALSE;
   diagStatus.axis.statusAxis.warning.bit20_Reserved := FALSE;
   diagStatus.axis.statusAxis.warning.bit21_Reserved := FALSE;
   diagStatus.axis.statusAxis.warning.bit22_Reserved := FALSE;
   diagStatus.axis.statusAxis.warning.bit23_Reserved := FALSE;
   diagStatus.axis.statusAxis.warning.bit24_Reserved := FALSE;
   diagStatus.axis.statusAxis.warning.bit25_Reserved := FALSE;
   diagStatus.axis.statusAxis.warning.bit26_Reserved := FALSE;
   diagStatus.axis.statusAxis.warning.bit27_Reserved := FALSE;
   diagStatus.axis.statusAxis.warning.bit28_Reserved := FALSE;
   diagStatus.axis.statusAxis.warning.bit29_Reserved := FALSE;
   diagStatus.axis.statusAxis.warning.bit30_Reserved := FALSE;
   diagStatus.axis.statusAxis.warning.bit31_Reserved := FALSE;
   diagStatus.axis.statusAxis.error.bit00_SystemFault := FALSE;
   diagStatus.axis.statusAxis.error.bit01_ConfigFault := FALSE;
   diagStatus.axis.statusAxis.error.bit02_UserFault := FALSE;
   diagStatus.axis.statusAxis.error.bit03_CommandNotAccepted := FALSE;
   diagStatus.axis.statusAxis.error.bit04_DriveFault := FALSE;
   diagStatus.axis.statusAxis.error.bit05_SensorFault := FALSE;
   diagStatus.axis.statusAxis.error.bit06_DynamicError := FALSE;
   diagStatus.axis.statusAxis.error.bit07_CommunicationFault := FALSE;
   diagStatus.axis.statusAxis.error.bit08_SWLimit := FALSE;
   diagStatus.axis.statusAxis.error.bit09_HWLimit := FALSE;
   diagStatus.axis.statusAxis.error.bit10_HomingError := FALSE;
   diagStatus.axis.statusAxis.error.bit11_FollowingErrorFault := FALSE;
   diagStatus.axis.statusAxis.error.bit12_PositioningFault := FALSE;
   diagStatus.axis.statusAxis.error.bit13_PeripheralError := FALSE;
   diagStatus.axis.statusAxis.error.bit14_SynchronousError := FALSE;
   diagStatus.axis.statusAxis.error.bit15_AdaptionError := FALSE;
   diagStatus.axis.statusAxis.error.bit16_Reserved := FALSE;
   diagStatus.axis.statusAxis.error.bit17_Reserved := FALSE;
   diagStatus.axis.statusAxis.error.bit18_Reserved := FALSE;
   diagStatus.axis.statusAxis.error.bit19_Reserved := FALSE;
   diagStatus.axis.statusAxis.error.bit20_Reserved := FALSE;
   diagStatus.axis.statusAxis.error.bit21_Reserved := FALSE;
   diagStatus.axis.statusAxis.error.bit22_Reserved := FALSE;
   diagStatus.axis.statusAxis.error.bit23_Reserved := FALSE;
   diagStatus.axis.statusAxis.error.bit24_Reserved := FALSE;
   diagStatus.axis.statusAxis.error.bit25_Reserved := FALSE;
   diagStatus.axis.statusAxis.error.bit26_Reserved := FALSE;
   diagStatus.axis.statusAxis.error.bit27_Reserved := FALSE;
   diagStatus.axis.statusAxis.error.bit28_Reserved := FALSE;
   diagStatus.axis.statusAxis.error.bit29_Reserved := FALSE;
   diagStatus.axis.statusAxis.error.bit30_Reserved := FALSE;
   diagStatus.axis.statusAxis.error.bit31_Reserved := FALSE;
   diagStatus.axis.statusAxis.errorDetail.number := 0;
   diagStatus.axis.statusAxis.errorDetail.reaction := 0;
   diagStatus.axis.statusSensor.operativeSensor := 1;
   diagStatus.axis.statusSensor.sensor[1..4].state := 0;
   diagStatus.axis.statusSensor.sensor[1..4].communicationOK := FALSE;
   diagStatus.axis.statusSensor.sensor[1..4].error := FALSE;
   diagStatus.axis.statusSensor.sensor[1..4].control := FALSE;
   diagStatus.axis.statusSensor.sensor[1..4].position := 0.0;
   diagStatus.axis.statusSensor.sensor[1..4].velocity := 0.0;
   diagStatus.axis.statusSensor.sensor[1..4].adaptionState := 0;
   diagStatus.axis.statusSensor.sensor[1..4].adjusted := 0;
   diagStatus.axis.statusPositioning.targetPosition := 0.0;
   diagStatus.axis.statusPositioning.followingError := 0.0;
   diagStatus.axis.units.lengthUnit := 0;
   diagStatus.axis.units.velocityUnit := 0;
   diagStatus.sina.sinaType := 0;
   diagStatus.sina.controlWord := 16#0000;
   diagStatus.sina.statusWord := 16#0000;
   diagStatus.sina.telegramNo := 0;
   diagStatus.sina.eposStatusWord1 := 16#0000;
   diagStatus.sina.eposStatusWord2 := 16#0000;
   diagStatus.sina.operatingDisplay := 0;
   diagStatus.sina.override := 0.0;
   diagStatus.sina.posSetValue := 0.0;
   diagStatus.sina.posActValue := 0.0;
   diagStatus.sina.velSetValue := 0.0;
   diagStatus.sina.velActValue := 0.0;
   diagStatus.sina.lengthUnit := 0;
   diagStatus.sina.velocityUnit := 0;
   diagStatus.sina.residualDistance := 0.0;
   diagStatus.sina.followingError := 0.0;
   diagStatus.sina.posControlWord := 16#0000;
   diagStatus.sina.posStatusWord := 16#0000;
   diagStatus.sina.blockSelected := 0;
   diagStatus.sina.blockActive := 0;
   diagStatus.sina.mdiPosSetValue := 0.0;
   diagStatus.sina.faultCode[0..7] := 16#0000;
   diagStatus.sina.alarmCode[0..3] := 16#0000;
   diagStatus.sina.speedSetValue := 0.0;
   diagStatus.sina.speedActValue := 0.0;
   diagStatus.sina.safetyStatusWord := 16#0000;
END_DATA_BLOCK

DATA_BLOCK "IdentData"   // DB221
TITLE = Schnittstelle Read/Write Daten / Interface read/write data
AUTHOR : SICAR
FAMILY : Ident
VERSION : 1.0
// Ident Daten / Ident data
// stored: MemoryReserve 100
   VAR
      rfReader { ExternalAccessible := 'False'; ExternalVisible := 'False'; ExternalWritable := 'False'} : Array[0.."NO_OF_RF_IDENT_DEVICES"] of "LSicar_typeIdentReadWriteDat";   // Reader
      mvReader { S7_SetPoint := 'True'} : Array[0.."NO_OF_MV_IDENT_DEVICES"] of "LSicar_typeIdentReadWriteDat";
   END_VAR
BEGIN
   rfReader[0].read[1..280] := 16#00;
   rfReader[1].read[1..280] := 16#00;
   rfReader[0].write[1..280] := 16#00;
   rfReader[1].write[1..280] := 16#00;
   mvReader[0].read[1..280] := 16#00;
   mvReader[1].read[1..280] := 16#00;
   mvReader[0].write[1..280] := 16#00;
   mvReader[1].write[1..280] := 16#00;
END_DATA_BLOCK

DATA_BLOCK "TestVarIdent"   // DB76
TITLE = Test tags fuer ident / Test tags for ident
AUTHOR : SICAR
FAMILY : Ident
VERSION : 1.0
// Test tags fuer ident / Test tags for ident
// stored: MemoryReserve 100
   VAR
      init1 : Bool := FALSE;   // Init 1
      read1 : Bool := FALSE;   // Read1
      write1 : Bool := FALSE;   // Write1
      init2 : Bool := FALSE;   // Init 2
      read2 : Bool := FALSE;   // Read2
      write2 : Bool := FALSE;   // Write2
      testString : String[32] := '';   // Test string
      charArr : Array[1..32] of Byte;   // Array of characters / Character Array
      prgNoMan : USInt := 0;   // Progrmm Nummer schreiben manual / Program number manual
      enableManCtrlRf : Bool := FALSE;   // Freigabe Manual Steuerung / Enable manual control RFID
      enableOption : Bool := FALSE;   // Freiegbae Optionen / Enable options
      enableManCtrlMV : Bool := FALSE;   // Enable manual control MV
   END_VAR
BEGIN
   charArr[1..32] := 16#00;
END_DATA_BLOCK

DATA_BLOCK "DiagnosticsSignalsInterface"   // DB138
// stored: MemoryReserve 100
   VAR
      SignalsInterface { S7_SetPoint := 'True'} : "LER_SignalsInterface";
   END_VAR
BEGIN
   SignalsInterface.HMI_Select_Mode := FALSE;
   SignalsInterface.ButtonValue[0].ButtonLeft[0..15] := FALSE;
   SignalsInterface.ButtonValue[1].ButtonLeft[0..15] := FALSE;
   SignalsInterface.ButtonValue[2].ButtonLeft[0..15] := FALSE;
   SignalsInterface.ButtonValue[3].ButtonLeft[0..15] := FALSE;
   SignalsInterface.ButtonValue[4].ButtonLeft[0..15] := FALSE;
   SignalsInterface.ButtonValue[5].ButtonLeft[0..15] := FALSE;
   SignalsInterface.ButtonValue[6].ButtonLeft[0..15] := FALSE;
   SignalsInterface.ButtonValue[7].ButtonLeft[0..15] := FALSE;
   SignalsInterface.ButtonValue[8].ButtonLeft[0..15] := FALSE;
   SignalsInterface.ButtonValue[9].ButtonLeft[0..15] := FALSE;
   SignalsInterface.ButtonValue[10].ButtonLeft[0..15] := FALSE;
   SignalsInterface.ButtonValue[11].ButtonLeft[0..15] := FALSE;
   SignalsInterface.ButtonValue[12].ButtonLeft[0..15] := FALSE;
   SignalsInterface.ButtonValue[13].ButtonLeft[0..15] := FALSE;
   SignalsInterface.ButtonValue[14].ButtonLeft[0..15] := FALSE;
   SignalsInterface.ButtonValue[15].ButtonLeft[0..15] := FALSE;
   SignalsInterface.ButtonValue[16].ButtonLeft[0..15] := FALSE;
   SignalsInterface.ButtonValue[0].ButtonRight[0..15] := FALSE;
   SignalsInterface.ButtonValue[1].ButtonRight[0..15] := FALSE;
   SignalsInterface.ButtonValue[2].ButtonRight[0..15] := FALSE;
   SignalsInterface.ButtonValue[3].ButtonRight[0..15] := FALSE;
   SignalsInterface.ButtonValue[4].ButtonRight[0..15] := FALSE;
   SignalsInterface.ButtonValue[5].ButtonRight[0..15] := FALSE;
   SignalsInterface.ButtonValue[6].ButtonRight[0..15] := FALSE;
   SignalsInterface.ButtonValue[7].ButtonRight[0..15] := FALSE;
   SignalsInterface.ButtonValue[8].ButtonRight[0..15] := FALSE;
   SignalsInterface.ButtonValue[9].ButtonRight[0..15] := FALSE;
   SignalsInterface.ButtonValue[10].ButtonRight[0..15] := FALSE;
   SignalsInterface.ButtonValue[11].ButtonRight[0..15] := FALSE;
   SignalsInterface.ButtonValue[12].ButtonRight[0..15] := FALSE;
   SignalsInterface.ButtonValue[13].ButtonRight[0..15] := FALSE;
   SignalsInterface.ButtonValue[14].ButtonRight[0..15] := FALSE;
   SignalsInterface.ButtonValue[15].ButtonRight[0..15] := FALSE;
   SignalsInterface.ButtonValue[16].ButtonRight[0..15] := FALSE;
END_DATA_BLOCK

DATA_BLOCK "TestVarMortorstarter"   // DB223
// stored: MemoryReserve 100
   VAR
      TestplantIdentifier : WString[24] := WSTRING#'++0.000MS1';
      faceplateType : USInt := 0;   // Bit for showing the buttons on FP
      operatorTripReset : Bool := FALSE;   // Operator Trip Reset Motorstarter
      contactorControlOn { S7_SetPoint := 'True'} : Bool := FALSE;
   END_VAR
BEGIN
END_DATA_BLOCK

DATA_BLOCK "OtherSafetyInterface"   // DB211
// stored: MemoryReserve 100
   VAR
      OtherDoor1 : "LER_typefDoorInterface";   // BA010 Other Door
      OtherDoor2 : "LER_typefDoorInterface";   // BA015 Other Door
      OtherDoor3 : "LER_typefDoorInterface";   // BA030 Other Door
      OtherDoor4 : "LER_typefDoorInterface";   // BA060 Other Door
      InspectionExternalDoor { S7_SetPoint := 'True'} : "LER_typefDoorInterface";   // Inspection External Door
      Inspection30MaintDoor { S7_SetPoint := 'True'} : "LER_typefDoorInterface";   // Inspection BA030 Main Door
      Inspection40MaintDoor { S7_SetPoint := 'True'} : "LER_typefDoorInterface";   // Inspection BA040 Main Door
      OtherEMO1 { S7_SetPoint := 'True'} : Bool;   // BA010 EMO
      OtherEMO2 { S7_SetPoint := 'True'} : Bool;   // BA015 EMO
      OtherEMO3 { S7_SetPoint := 'True'} : Bool;   // BA030 EMO
      OtherEMO4 { S7_SetPoint := 'True'} : Bool;   // BA060 EMO
      Inspection30LightCurtain { S7_SetPoint := 'True'} : "LER_typeLightCurtainInterface";   // BA060 Stack #1 Light Curatain
      Inspection40LightCurtain { S7_SetPoint := 'True'} : "LER_typeLightCurtainInterface";   // BA060 Stack #2 Light Curatain
      "30CathodeConveyorCover" { S7_SetPoint := 'True'} : "LER_typeConveyorCoverInterface";   // BA030 Cathode Conveyor Cover
      "30AnodeConveyorCover" { S7_SetPoint := 'True'} : "LER_typeConveyorCoverInterface";   // BA030 Cathode Anode Cover
      "40CathodeConveyorCover" { S7_SetPoint := 'True'} : "LER_typeConveyorCoverInterface";   // BA040 Cathode Conveyor Cover
      "40AnodeConveyorCover" { S7_SetPoint := 'True'} : "LER_typeConveyorCoverInterface";   // BA040 Cathode Anode Cover
   END_VAR
BEGIN
   OtherDoor1.configuration.referenceDesignator := WSTRING#'10';
   OtherDoor2.configuration.referenceDesignator := WSTRING#'15';
   OtherDoor3.configuration.referenceDesignator := WSTRING#'30';
   OtherDoor4.configuration.referenceDesignator := WSTRING#'60';
   InspectionExternalDoor.configuration.referenceDesignator := WSTRING#'60';
   Inspection30MaintDoor.configuration.referenceDesignator := WSTRING#'30';
   Inspection40MaintDoor.configuration.referenceDesignator := WSTRING#'40';
   Inspection30LightCurtain.configuration.referenceDesignator := WSTRING#'30';
   Inspection40LightCurtain.configuration.referenceDesignator := WSTRING#'40';
   "30CathodeConveyorCover".configuration.referenceDesignator := WSTRING#'30-CA';
   "30AnodeConveyorCover".configuration.referenceDesignator := WSTRING#'30-AN';
   "40CathodeConveyorCover".configuration.referenceDesignator := WSTRING#'40-CA';
   "40AnodeConveyorCover".configuration.referenceDesignator := WSTRING#'40-AN';
END_DATA_BLOCK

DATA_BLOCK "Safetyinterface"   // DB256
// stored: MemoryReserve 100
   VAR
      StackDoor1 : "LER_typefDoorInterface";
      StackDoor2 : "LER_typefDoorInterface";
      StackDoor3 : "LER_typefDoorInterface";
      StackDoor4 : "LER_typefDoorInterface";
      StackDoor5 : "LER_typefDoorInterface";
      StackDoor6 : "LER_typefDoorInterface";
      StackDoor7 : "LER_typefDoorInterface";
      StackDoor8 : "LER_typefDoorInterface";
      StackDoor9 : "LER_typefDoorInterface";
      StackDoor10 : "LER_typefDoorInterface";
      StackDoor11 : "LER_typefDoorInterface";
      StackDoor12 : "LER_typefDoorInterface";
   END_VAR
BEGIN
   StackDoor1.commands.Lock := FALSE;
   StackDoor1.commands.Unlock := FALSE;
   StackDoor1.monitoring.DoorOpen := FALSE;
   StackDoor1.monitoring.DoorClose := TRUE;
   StackDoor1.monitoring.DoorLock := TRUE;
   StackDoor1.monitoring.DoorUnLock := FALSE;
   StackDoor1.configuration.referenceDesignator := WSTRING#'AUTO SPL';
   StackDoor2.commands.Lock := FALSE;
   StackDoor2.commands.Unlock := FALSE;
   StackDoor2.monitoring.DoorOpen := FALSE;
   StackDoor2.monitoring.DoorClose := TRUE;
   StackDoor2.monitoring.DoorLock := TRUE;
   StackDoor2.monitoring.DoorUnLock := FALSE;
   StackDoor2.configuration.referenceDesignator := WSTRING#'U/W MAIN';
   StackDoor3.commands.Lock := FALSE;
   StackDoor3.commands.Unlock := FALSE;
   StackDoor3.monitoring.DoorOpen := FALSE;
   StackDoor3.monitoring.DoorClose := TRUE;
   StackDoor3.monitoring.DoorLock := TRUE;
   StackDoor3.monitoring.DoorUnLock := FALSE;
   StackDoor3.configuration.referenceDesignator := WSTRING#'U/W TOP';
   StackDoor4.commands.Lock := FALSE;
   StackDoor4.commands.Unlock := FALSE;
   StackDoor4.monitoring.DoorOpen := FALSE;
   StackDoor4.monitoring.DoorClose := TRUE;
   StackDoor4.monitoring.DoorLock := TRUE;
   StackDoor4.monitoring.DoorUnLock := FALSE;
   StackDoor4.configuration.referenceDesignator := WSTRING#'U/W BTM';
   StackDoor5.commands.Lock := FALSE;
   StackDoor5.commands.Unlock := FALSE;
   StackDoor5.monitoring.DoorOpen := FALSE;
   StackDoor5.monitoring.DoorClose := TRUE;
   StackDoor5.monitoring.DoorLock := TRUE;
   StackDoor5.monitoring.DoorUnLock := FALSE;
   StackDoor5.configuration.referenceDesignator := WSTRING#'TBL FRNT';
   StackDoor6.commands.Lock := FALSE;
   StackDoor6.commands.Unlock := FALSE;
   StackDoor6.monitoring.DoorOpen := FALSE;
   StackDoor6.monitoring.DoorClose := TRUE;
   StackDoor6.monitoring.DoorLock := TRUE;
   StackDoor6.monitoring.DoorUnLock := FALSE;
   StackDoor6.configuration.referenceDesignator := WSTRING#'WINDER';
   StackDoor7.commands.Lock := FALSE;
   StackDoor7.commands.Unlock := FALSE;
   StackDoor7.monitoring.DoorOpen := FALSE;
   StackDoor7.monitoring.DoorClose := TRUE;
   StackDoor7.monitoring.DoorLock := TRUE;
   StackDoor7.monitoring.DoorUnLock := FALSE;
   StackDoor7.configuration.referenceDesignator := WSTRING#'A-WASTE';
   StackDoor8.commands.Lock := FALSE;
   StackDoor8.commands.Unlock := FALSE;
   StackDoor8.monitoring.DoorOpen := FALSE;
   StackDoor8.monitoring.DoorClose := TRUE;
   StackDoor8.monitoring.DoorLock := TRUE;
   StackDoor8.monitoring.DoorUnLock := FALSE;
   StackDoor8.configuration.referenceDesignator := WSTRING#'TBL REAR';
   StackDoor9.commands.Lock := FALSE;
   StackDoor9.commands.Unlock := FALSE;
   StackDoor9.monitoring.DoorOpen := FALSE;
   StackDoor9.monitoring.DoorClose := TRUE;
   StackDoor9.monitoring.DoorLock := TRUE;
   StackDoor9.monitoring.DoorUnLock := FALSE;
   StackDoor9.configuration.referenceDesignator := WSTRING#'C-WASTE';
   StackDoor10.commands.Lock := FALSE;
   StackDoor10.commands.Unlock := FALSE;
   StackDoor10.monitoring.DoorOpen := FALSE;
   StackDoor10.monitoring.DoorClose := TRUE;
   StackDoor10.monitoring.DoorLock := TRUE;
   StackDoor10.monitoring.DoorUnLock := FALSE;
   StackDoor10.configuration.referenceDesignator := WSTRING#'U/W REAR';
   StackDoor11.commands.Lock := FALSE;
   StackDoor11.commands.Unlock := FALSE;
   StackDoor11.monitoring.DoorOpen := FALSE;
   StackDoor11.monitoring.DoorClose := TRUE;
   StackDoor11.monitoring.DoorLock := TRUE;
   StackDoor11.monitoring.DoorUnLock := FALSE;
   StackDoor11.configuration.referenceDesignator := WSTRING#'';
   StackDoor12.commands.Lock := FALSE;
   StackDoor12.commands.Unlock := FALSE;
   StackDoor12.monitoring.DoorOpen := FALSE;
   StackDoor12.monitoring.DoorClose := TRUE;
   StackDoor12.monitoring.DoorLock := TRUE;
   StackDoor12.monitoring.DoorUnLock := FALSE;
   StackDoor12.configuration.referenceDesignator := WSTRING#'';
END_DATA_BLOCK

DATA_BLOCK "ProdDataSimulation"   // DB5
{ DB_Accessible_From_OPC_UA := 'FALSE' }
// stored: DBAccessibleFromOPCUA false, DBAccessibleFromWebserver false, MemoryReserve 100
   VAR
      ProdDataCounter { ExternalAccessible := 'False'; ExternalVisible := 'False'; ExternalWritable := 'False'} : Struct   // Test tag prod data
         ProdDataCounter1Up1 : Bool := FALSE;   // Test Variable Prod. Daten / Test tag prod data
         ProdDataCounter1Up2 : Bool := FALSE;   // Test Variable Prod. Daten / Test tag prod data
         ProdDataCounter1Down1 : Bool := FALSE;   // Test Variable Prod. Daten / Test tag prod data
         ProdDataCounter1Down2 : Bool := FALSE;   // Test Variable Prod. Daten / Test tag prod data
         ProdDataCounter1Reset1 : Bool := FALSE;   // Test Variable Prod. Daten / Test tag prod data
         ProdDataCounter1Reset2 : Bool := FALSE;   // Test Variable Prod. Daten / Test tag prod data
         ProdDataCounter1ResetAll : Bool := FALSE;   // Test Variable Prod. Daten / Test tag prod data
         ProdDataCounter2Up1 : Bool := FALSE;
         ProdDataCounter2Up2 : Bool := FALSE;
         ProdDataCounter2Down1 : Bool := FALSE;
         ProdDataCounter2Down2 : Bool := FALSE;
         ProdDataCounter2Reset1 : Bool := FALSE;
         ProdDataCounter2Reset2 : Bool := FALSE;
         ProdDataCounter2ResetAll : Bool := FALSE;
         userInterfaceVisibilityDataSet2Counter : DWord := 16#000F_FFFF;
         userInterfaceVisibilityDataSet1Counter : DWord := 16#0000_3FFF;
         ProdDataEnable : Bool := FALSE;
      END_STRUCT;
      ProdDataCyclic { ExternalAccessible := 'False'; ExternalVisible := 'False'; ExternalWritable := 'False'} : Struct   // Test tag prod data
         cycleTimer1Run1 : Bool := FALSE;   // Test Variable Prod. Daten / Test tag prod data
         cycleTimer1Run2 : Bool := FALSE;   // Test Variable Prod. Daten / Test tag prod data
         cycleTimer1Hold1 : Bool := FALSE;   // Test Variable Prod. Daten / Test tag prod data
         cycleTimer1Hold2 : Bool := FALSE;   // Test Variable Prod. Daten / Test tag prod data
         cycleTimer1Reset1 : Bool := FALSE;   // Test Variable Prod. Daten / Test tag prod data
         cycleTimer1Reset2 : Bool := FALSE;   // Test Variable Prod. Daten / Test tag prod data
         cycleTimer1ResetAll : Bool := FALSE;   // Test Variable Prod. Daten / Test tag prod data
         cycleTimer2Run1 : Bool := FALSE;   // Test Variable Prod. Daten / Test tag prod data
         cycleTimer2Run2 : Bool := FALSE;   // Test Variable Prod. Daten / Test tag prod data
         cycleTimer2Hold1 : Bool := FALSE;   // Test Variable Prod. Daten / Test tag prod data
         cycleTimer2Hold2 : Bool := FALSE;   // Test Variable Prod. Daten / Test tag prod data
         cycleTimer2Reset1 : Bool := FALSE;   // Test Variable Prod. Daten / Test tag prod data
         cycleTimer2Reset2 : Bool := FALSE;   // Test Variable Prod. Daten / Test tag prod data
         cycleTimer2ResetAll : Bool := FALSE;   // Test Variable Prod. Daten / Test tag prod data
         cyclicTimerEnable : Bool := FALSE;
         userInterfaceVisibilityDataSet2Cyclic : DWord := 2#0000_0000_0000_0000_0000_0010_0000_0011;
         userInterfaceVisibilityDataSet1Cyclic : DWord := 2#0000_0000_0000_0000_0000_0010_0000_0011;
         userInterfaceVisibilityDataSet3Cyclic : DWord := 2#0000_0000_0000_0000_0000_0010_0000_0011;
         userInterfaceVisibilityDataSet4Cyclic : DWord := 2#0000_0000_0000_0000_0000_0000_0000_0011;
         userInterfaceVisibilityDataSet5Cyclic : DWord := 2#0000_0000_0000_0001_1111_1111_1011_1111;
         userInterfaceVisibilityDataSet6Cyclic : DWord := 2#0000_0000_0000_0001_1111_1111_1011_1111;
         userInterfaceVisibilityDataSet7Cyclic : DWord := 2#0000_0000_0000_0101_0011_1100_1100_1011;
         userInterfaceVisibilityDataSet8Cyclic : DWord := 2#0000_0000_0000_0000_1111_1101_1111_0111;
      END_STRUCT;
      ProdDataLimitValues { ExternalAccessible := 'False'; ExternalVisible := 'False'; ExternalWritable := 'False'} : Struct   // Test tag prod data
         limitVal1Count1PreWarn1 : Bool := FALSE;   // Test Variable Prod. Daten / Test tag prod data
         limitVal1Count1PreWarn3 : Bool := FALSE;   // Test Variable Prod. Daten / Test tag prod data
         limitVal1Count1PreWarn2 : Bool := FALSE;   // Test Variable Prod. Daten / Test tag prod data
         limitVal1Count1Alarm1 : Bool := FALSE;   // Test Variable Prod. Daten / Test tag prod data
         limitVal1Count1Alarm3 : Bool := FALSE;   // Test Variable Prod. Daten / Test tag prod data
         limitVal1Count1Alarm2 : Bool := FALSE;   // Test Variable Prod. Daten / Test tag prod data
         limitVal1Count1 : Bool := FALSE;   // Test Variable Prod. Daten / Test tag prod data
         limitVal1Count2 : Bool := FALSE;   // Test Variable Prod. Daten / Test tag prod data
         limitVal1Count3 : Bool := FALSE;   // Test Variable Prod. Daten / Test tag prod data
         limitVal1Set1 : Bool := FALSE;   // Test Variable Prod. Daten / Test tag prod data
         limitVal1Set3 : Bool := FALSE;   // Test Variable Prod. Daten / Test tag prod data
         limitVal1Set2 : Bool := FALSE;   // Test Variable Prod. Daten / Test tag prod data
         limitValuesEnable : Bool := FALSE;
         userInterfaceVisibilityDataSet2LimitValues : DWord := 16#0000_03FF;
         userInterfaceVisibilityDataSet1LimitValues : DWord := 16#0000_000F;
      END_STRUCT;
      ProdDataShiftCounter { ExternalAccessible := 'False'; ExternalVisible := 'False'; ExternalWritable := 'False'} : Struct   // Test tag prod data
         shiftCounter1Cnt1Curr : Bool := FALSE;   // Test Variable Prod. Daten / Test tag prod data
         shiftCounter1Cnt1CurrOk : Bool := FALSE;   // Test Variable Prod. Daten / Test tag prod data
         shiftCounter1Cnt2Curr : Bool := FALSE;   // Test Variable Prod. Daten / Test tag prod data
         shiftCounter1Cnt2CurrOk : Bool := FALSE;   // Test Variable Prod. Daten / Test tag prod data
         shiftCounter1Cnt3Curr : Bool := FALSE;   // Test Variable Prod. Daten / Test tag prod data
         shiftCounter1Cnt3CurrOk : Bool := FALSE;   // Test Variable Prod. Daten / Test tag prod data
         shiftCounter1ResetAllExt : Bool := FALSE;   // Test Variable Prod. Daten / Test tag prod data
         ShiftCounterEnable : Bool := FALSE;
         userInterfaceVisibilityDataSet2ShiftCounter : DWord := 16#0000_03FF;
         userInterfaceVisibilityDataSet1ShiftCounter : DWord := 16#0000_000F;
      END_STRUCT;
      ProdDataShiftCounterOEE { ExternalAccessible := 'False'; ExternalVisible := 'False'; ExternalWritable := 'False'} : Struct   // Test tag prod data
         ShiftCounterOEEEnable : Bool := FALSE;
         userInterfaceVisibilityDataSet2ShiftCounterOEE : DWord := 16#0000_03FF;
         userInterfaceVisibilityDataSet1ShiftCounterOEE : DWord := 16#0000_000F;
      END_STRUCT;
   END_VAR
BEGIN
END_DATA_BLOCK

DATA_BLOCK "PM01"   // DB334
// stored: MemoryReserve 100
   VAR
      "SEPA DANCER FORWARD" : Bool := FALSE;
      "SEPA DANCER BACKWARD" : Bool := FALSE;
      "SEPA UW #1 IONIZER TOP ON" : Bool := FALSE;
      SPARE : Bool := FALSE;
      "SEPA UW #1 IONIZER BTM ON" : Bool := FALSE;
      SPARE_1 : Bool := FALSE;
      "SEPA UW #1 AIR SHAFT TOP ON" : Bool := FALSE;
      "SEPA UW #1 AIR SHAFT TOP OFF" : Bool := FALSE;
      "SEPA UW #1 AIR SHAFT BTM ON" : Bool := FALSE;
      "SEPA UW #1 AIR SHAFT BTM OFF" : Bool := FALSE;
      SPARE_3 : Bool := FALSE;
      SPARE_4 : Bool := FALSE;
      "ANODE CONVEYOR PICK UP BLOWER ON/OFF" : Bool := FALSE;
      SPARE_2 : Bool := FALSE;
      "CATHODE CONVEYOR PICK UP BLOWER ON/OFF" : Bool := FALSE;
   END_VAR
BEGIN
END_DATA_BLOCK

DATA_BLOCK "PM02"   // DB336
// stored: MemoryReserve 100
   VAR
      "SUCTION PAD #1 TOP UP" : Bool := FALSE;
      "SUCTION PAD #1 TOP DOWN" : Bool := FALSE;
      "SUCTION PAD #1 BTM UP" : Bool := FALSE;
      "SUCTION PAD #1 BTM DOWN" : Bool := FALSE;
      "CUTTER #1 UP" : Bool := FALSE;
      "CUTTER #1 DOWN" : Bool := FALSE;
      "TAPE #1 TOP UP" : Bool := FALSE;
      "TAPE #1 TOP DOWN" : Bool := FALSE;
      "TAPE #1 BTM UP" : Bool := FALSE;
      "TAPE #1 BTM DOWN" : Bool := FALSE;
      "SPLICE HEAD ROTATE #1 TOP FORWARD" : Bool := FALSE;
      "SPLICE HEAD ROTATE #1 TOP BACKWARD" : Bool := FALSE;
      "SPLICE HEAD ROTATE #1 BTM FORWARD" : Bool := FALSE;
      "SPLICE HEAD ROTATE #1 BTM BACKWARD" : Bool := FALSE;
   END_VAR
BEGIN
END_DATA_BLOCK

DATA_BLOCK "PM03"   // DB338
// stored: MemoryReserve 100
   VAR
      "SEPA CUTTER REAR UP / SEPA CUTTER FRONT UP" : Bool := FALSE;
      "SEPA CUTTER REAR DOWN / SEPA CUTTER FRONT DOWN" : Bool := FALSE;
      "SEPA CLAMP TOP REAR UP" : Bool := FALSE;
      "SEPA CLAMP TOP REAR DOWN" : Bool := FALSE;
      "SEPA CLAMP TOP FRONT UP" : Bool := FALSE;
      "SEPA CLAMP TOP FRONT DOWN" : Bool := FALSE;
      "SEPA CLAMP BTM REAR UP" : Bool := FALSE;
      "SEPA CLAMP BTM REAR DOWN" : Bool := FALSE;
      "SEPA CLAMP BTM FRONT UP" : Bool := FALSE;
      "SEPA CLAMP BTM FRONT DOWN" : Bool := FALSE;
      "SEPA GRIPPER OPEN" : Bool := FALSE;
      "SEPA GRIPPER  CLOSE" : Bool := FALSE;
      "SEPA GRIPPER FORWARD" : Bool := FALSE;
      "SEPA GRIPPER BACKWARD" : Bool := FALSE;
   END_VAR
BEGIN
END_DATA_BLOCK

DATA_BLOCK "PM04"   // DB337
// stored: MemoryReserve 100
   VAR
      "STACK TABLE GAP PAD UP" : Bool := FALSE;
      "STACK TABLE GAP PAD DOWN" : Bool := FALSE;
      "CATHODE MANDREL CLAMP FRONT ON" : Bool := FALSE;
      SPARE : Bool := FALSE;
      "CATHODE MANDREL CLAMP REAR ON" : Bool := FALSE;
      SPARE_1 : Bool := FALSE;
      "ANODE MANDREL CLAMP FRONT ON" : Bool := FALSE;
      SPARE_2 : Bool := FALSE;
      "ANODE MANDREL CLAMP REAR ON" : Bool := FALSE;
   END_VAR
BEGIN
END_DATA_BLOCK

DATA_BLOCK "PM05"   // DB233
// stored: MemoryReserve 100
   VAR
      "ANODE GLASS CLEANING ON" : Bool := FALSE;
      SPARE : Bool := FALSE;
      "ANODE MAIN NG P&P UP" : Bool := FALSE;
      "ANODE MAIN NG P&P DOWN" : Bool := FALSE;
      "ANODE MAIN NG P&P 1st FORWARD" : Bool := FALSE;
      "ANODE MAIN NG P&P 1st BACKWARD" : Bool := FALSE;
      "ANODE MAIN NG P&P 2nd FORWARD" : Bool := FALSE;
      "ANODE MAIN NG P&P 2nd BACKWARD" : Bool := FALSE;
      "ANODE FIX FRONT FORWARD / ANODE FIX REAR FORWARD" : Bool := FALSE;
      "ANODE FIX FRONT BACKWARD / ANODE FIX REAR BACKWARD" : Bool := FALSE;
      "ANODE MAIN P&P#1 Rotary CW" : Bool := FALSE;
      "ANODE MAIN P&P#1 Rotary CCW" : Bool := FALSE;
      "ANODE NG BOX LIFT UP" : Bool := FALSE;
      "ANODE NG BOX LIFT DOWN" : Bool := FALSE;
      "ANODE NG BOX LOCK UP" : Bool := FALSE;
      "ANODE NG BOX LOCK DOWN" : Bool := FALSE;
   END_VAR
BEGIN
END_DATA_BLOCK

DATA_BLOCK "PM06"   // DB335
// stored: MemoryReserve 100
   VAR
      "CATHODE GLASS CLEANING ON" : Bool := FALSE;
      SPARE : Bool := FALSE;
      "CATHODE MAIN NG P&P UP" : Bool := FALSE;
      "CATHODE MAIN NG P&P DOWN" : Bool := FALSE;
      "CATHODE MAIN NG P&P 1st FORWARD" : Bool := FALSE;
      "CATHODE MAIN NG P&P 1st BACKWARD" : Bool := FALSE;
      "CATHODE MAIN NG P&P 2nd FORWARD" : Bool := FALSE;
      "CATHODE MAIN NG P&P 2nd BACKWARD" : Bool := FALSE;
      "CATHODE FIX FRONT FORWARD / CATHODE FIX REAR FORWARD" : Bool := FALSE;
      "CATHODE FIX FRONT BACKWARD / CATHODE FIX REAR BACKWARD" : Bool := FALSE;
      "CATHODE MAIN P&P#1 Rotary CW" : Bool := FALSE;
      "CATHODE MAIN P&P#1 Rotary CCW" : Bool := FALSE;
      "CATHODE NG BOX LIFT UP" : Bool := FALSE;
      "CATHODE NG BOX LIFT DOWN" : Bool := FALSE;
      "CATHODE NG BOX LOCK UP" : Bool := FALSE;
      "CATHODE NG BOX LOCK DOWN" : Bool := FALSE;
   END_VAR
BEGIN
END_DATA_BLOCK

DATA_BLOCK "PM07"   // DB333
// stored: MemoryReserve 100
   VAR
      "JR WINDER CLAMP TOP REAR  UP" : Bool := FALSE;
      "JR WINDER CLAMP TOP REAR  DOWN" : Bool := FALSE;
      "JR WINDER CLAMP BTM REAR UP" : Bool := FALSE;
      "JR WINDER CLAMP BTM REAR DOWN" : Bool := FALSE;
      "JR WINDER CLAMP TOP FRONT UP" : Bool := FALSE;
      "JR WINDER CLAMP TOP FRONT DOWN" : Bool := FALSE;
      "JR WINDER CLAMP BTM FRONT UP" : Bool := FALSE;
      "JR WINDER CLAMP BTM FRONT DOWN" : Bool := FALSE;
      SPARE : Bool := FALSE;
      SPARE_1 : Bool := FALSE;
      "PUSH ROLLER FORWARD" : Bool := FALSE;
      "PUSH ROLLER BACKWARD" : Bool := FALSE;
      "ANODE CONVEYOR COVER FORWARD" : Bool := FALSE;
      "ANODE CONVEYOR COVER BACKWARD" : Bool := FALSE;
      "CATHODE CONVEYOR COVER FORWARD" : Bool := FALSE;
      "CATHODE CONVEYOR COVER BACKWARD" : Bool := FALSE;
   END_VAR
BEGIN
END_DATA_BLOCK

DATA_BLOCK "SBK01"   // DB322
// stored: MemoryReserve 100
   VAR
      "EMO01 CH.A" : Bool;
      "EMO02 CH.A" : Bool;
      SPARE : Bool;
      "EMO04 CH.A" : Bool;
      "EMO01 CH.B" : Bool;
      "EMO02 CH.B" : Bool;
      SPARE_1 : Bool;
      "EMO04 CH.B" : Bool;
      SPARE_2 : Bool;
      SPARE_3 : Bool;
      SPARE_4 : Bool;
   END_VAR
BEGIN
END_DATA_BLOCK

DATA_BLOCK "SBK02"   // DB323
// stored: MemoryReserve 100
   VAR
      "SCS BOX SCS MODE SLELECT SS.SETUP" : Bool := FALSE;
      "SCS BOX SCS MODE SLELECT SS.DISABLE" : Bool := FALSE;
      "EMO05 CH.A" : Bool := FALSE;
      SPARE : Bool := FALSE;
      "SCS BOX SCS MODE SLELECT SS.AUTO" : Bool := TRUE;
      SPARE_1 : Bool := FALSE;
      "EMO05 CH.B" : Bool := FALSE;
      SPARE_2 : Bool := FALSE;
      "SCS BOX SCS MODE SELECT PL.PENDANT" : Bool := FALSE;
      "SCS BOX SCS MODE SELECT PL.DISABLE" : Bool := FALSE;
      SPARE_3 : Bool;
   END_VAR
BEGIN
END_DATA_BLOCK

DATA_BLOCK "SBK03"   // DB317
// stored: MemoryReserve 100
   VAR
      "ROLL CHANGE TOP SS.AUTO" : Bool := TRUE;
      "ROLL CHANGE BTM SS.AUTO" : Bool := TRUE;
      SPARE : Bool := FALSE;
      SPARE_1 : Bool := FALSE;
      "ROLL CHANGE TOP SS.CHANGE" : Bool := FALSE;
      "ROLL CHANGE BTM SS.CHANGE" : Bool := FALSE;
      SPARE_2 : Bool := FALSE;
      SPARE_3 : Bool := FALSE;
      "ROLL CHANGE LH IN PROGRESS" : Bool := FALSE;
      "ROLL CHANGE RH IN PROGRESS" : Bool := FALSE;
      SPARE_4 : Bool;
   END_VAR
BEGIN
END_DATA_BLOCK

DATA_BLOCK "SBK04"   // DB319
// stored: MemoryReserve 100
   VAR
      "GATE EC U/W MAIN PB.LOCK" : Bool := FALSE;
      "GATE EC U/W MAIN PB.RESET" : Bool := FALSE;
      SPARE : Bool := FALSE;
      SPARE_1 : Bool := FALSE;
      "GATE EC U/W MAIN PB.UNLOCK" : Bool := FALSE;
      SPARE_2 : Bool := FALSE;
      SPARE_3 : Bool := FALSE;
      SPARE_4 : Bool := FALSE;
      "GATE EC U/W MAIN PL.LOCK" : Bool := TRUE;
      "GATE EC U/W MAIN PL.UNLOCK" : Bool := FALSE;
      "GATE EC U/W MAIN PL.RESET" : Bool := TRUE;
   END_VAR
BEGIN
END_DATA_BLOCK

DATA_BLOCK "SBK05"   // DB318
// stored: MemoryReserve 100
   VAR
      "GATE EC U/W TOP PB.LOCK" : Bool := FALSE;
      "GATE EC U/W TOP PB.RESET" : Bool := FALSE;
      SPARE : Bool := FALSE;
      SPARE_1 : Bool := FALSE;
      "GATE EC U/W TOP PB.UNLOCK" : Bool := FALSE;
      SPARE_2 : Bool := FALSE;
      SPARE_3 : Bool := FALSE;
      SPARE_4 : Bool := FALSE;
      "GATE EC U/W TOP PL.LOCK" : Bool := TRUE;
      "GATE EC U/W TOP PL.UNLOCK" : Bool := FALSE;
      "GATE EC U/W TOP PL.RESET" : Bool := TRUE;
   END_VAR
BEGIN
END_DATA_BLOCK

DATA_BLOCK "SBK06"   // DB202
// stored: MemoryReserve 100
   VAR
      "GATE EC U/W BTM PB.LOCK" : Bool := FALSE;
      "GATE EC U/W BTM PB.RESET" : Bool := FALSE;
      SPARE : Bool := FALSE;
      SPARE_1 : Bool := FALSE;
      "GATE EC U/W BTM PB.UNLOCK" : Bool := FALSE;
      SPARE_2 : Bool := FALSE;
      SPARE_3 : Bool := FALSE;
      SPARE_4 : Bool := FALSE;
      "GATE EC U/W BTM PL.LOCK" : Bool := TRUE;
      "GATE EC U/W BTM PL.UNLOCK" : Bool := TRUE;
      "GATE EC U/W BTM PL.RESET" : Bool := TRUE;
   END_VAR
BEGIN
END_DATA_BLOCK

DATA_BLOCK "SBK07"   // DB320
// stored: MemoryReserve 100
   VAR
      "GATE EC SCRAP BOX-1 PB.LOCK" : Bool := FALSE;
      "GATE EC SCRAP BOX-1 PB.RESET" : Bool := FALSE;
      SPARE : Bool := FALSE;
      SPARE_1 : Bool := FALSE;
      "GATE EC SCRAP BOX-1 PB.UNLOCK" : Bool := FALSE;
      SPARE_2 : Bool := FALSE;
      SPARE_3 : Bool := FALSE;
      SPARE_4 : Bool := FALSE;
      "GATE EC SCRAP BOX-1 PL.LOCK" : Bool := FALSE;
      "GATE EC SCRAP BOX-1 PL.UNLOCK" : Bool := TRUE;
      "GATE EC SCRAP BOX-1 PL.RESET" : Bool := FALSE;
   END_VAR
BEGIN
END_DATA_BLOCK

DATA_BLOCK "SBK08"   // DB321
// stored: MemoryReserve 100
   VAR
      "SAFETY DOOR LOCK1.INPUT" : Bool := TRUE;
      "SAFETY DOOR LOCK2.INPUT" : Bool := TRUE;
      "SAFETY DOOR LOCK3.INPUT" : Bool := TRUE;
      SPARE : Bool := FALSE;
      "SAFETY DOOR LOCK1.INPUT_1" : Bool := FALSE;
      "SAFETY DOOR LOCK2.INPUT_1" : Bool := FALSE;
      "SAFETY DOOR LOCK3.INPUT_1" : Bool := FALSE;
      SPARE_1 : Bool := FALSE;
      "SAFETY DOOR LOCK1.OUTPUT" : Bool := FALSE;
      "SAFETY DOOR LOCK2.OUTPUT" : Bool := FALSE;
      "SAFETY DOOR LOCK3.OUTPUT" : Bool := FALSE;
   END_VAR
BEGIN
END_DATA_BLOCK

DATA_BLOCK "SBK09"   // DB326
// stored: MemoryReserve 100
   VAR
      "SAFETY DOOR LOCK4.INPUT" : Bool := TRUE;
      "SAFETY DOOR LOCK5.INPUT" : Bool := TRUE;
      "SAFETY DOOR LOCK6.INPUT" : Bool := TRUE;
      SPARE : Bool := FALSE;
      "SAFETY DOOR LOCK4.INPUT_1" : Bool := FALSE;
      "SAFETY DOOR LOCK5.INPUT_1" : Bool := FALSE;
      "SAFETY DOOR LOCK6.INPUT_1" : Bool := FALSE;
      SPARE_1 : Bool := FALSE;
      "SAFETY DOOR LOCK4.OUTPUT" : Bool := FALSE;
      "SAFETY DOOR LOCK5.OUTPUT" : Bool := FALSE;
      "SAFETY DOOR LOCK6.OUTPUT" : Bool := FALSE;
   END_VAR
BEGIN
END_DATA_BLOCK

DATA_BLOCK "SBK10"   // DB328
// stored: MemoryReserve 100
   VAR
      "SAFETY DOOR LOCK7.INPUT" : Bool := TRUE;
      "SAFETY DOOR LOCK8.INPUT" : Bool := TRUE;
      SPARE : Bool := TRUE;
      SPARE_1 : Bool := FALSE;
      "SAFETY DOOR LOCK7.INPUT_1" : Bool := FALSE;
      "SAFETY DOOR LOCK8.INPUT_1" : Bool := FALSE;
      SPARE_2 : Bool := FALSE;
      SPARE_3 : Bool := FALSE;
      "SAFETY DOOR LOCK7.OUTPUT" : Bool := FALSE;
      "SAFETY DOOR LOCK8.OUTPUT" : Bool := FALSE;
      SPARE_4 : Bool := FALSE;
   END_VAR
BEGIN
END_DATA_BLOCK

DATA_BLOCK "SBK11"   // DB324
// stored: MemoryReserve 100
   VAR
      "GATE EC SCRAP BOX-2 PB.LOCK" : Bool := FALSE;
      "GATE EC SCRAP BOX-2 PB.RESET" : Bool := FALSE;
      SPARE : Bool := FALSE;
      SPARE_1 : Bool := FALSE;
      "GATE EC SCRAP BOX-2 PB.UNLOCK" : Bool := FALSE;
      SPARE_2 : Bool := FALSE;
      SPARE_3 : Bool := FALSE;
      SPARE_4 : Bool := FALSE;
      "GATE EC SCRAP BOX-2 PL.LOCK" : Bool := FALSE;
      "GATE EC SCRAP BOX-2 PL.UNLOCK" : Bool := TRUE;
      "GATE EC SCRAP BOX-2 PL.RESET" : Bool := FALSE;
   END_VAR
BEGIN
END_DATA_BLOCK

DATA_BLOCK "SBK12"   // DB325
// stored: MemoryReserve 100
   VAR
      "ANODE CONVEYOR COVER BACKWARD" : Bool := FALSE;
      "CATHODE CONVEYOR COVER BACKWARD" : Bool := FALSE;
      SPARE : Bool := FALSE;
      SPARE_1 : Bool := FALSE;
      "ANODE CONVEYOR COVER FORWARD" : Bool := FALSE;
      "CATHODE CONVEYOR COVER FORWARD" : Bool := FALSE;
      SPARE_2 : Bool := FALSE;
      SPARE_3 : Bool := FALSE;
      SPARE_4 : Bool;
      SPARE_5 : Bool;
      SPARE_6 : Bool;
   END_VAR
BEGIN
END_DATA_BLOCK

DATA_BLOCK "SBK13"   // DB327
// stored: MemoryReserve 100
   VAR
      "SAFETY DOOR LOCK10.INPUT" : Bool := FALSE;
      SPARE : Bool := FALSE;
      "SAFETY DOOR LOCK12.INPUT" : Bool := FALSE;
      SPARE_1 : Bool := FALSE;
      "SAFETY DOOR LOCK10.INPUT_1" : Bool := FALSE;
      SPARE_2 : Bool := FALSE;
      "SAFETY DOOR LOCK12.INPUT_1" : Bool := FALSE;
      SPARE_3 : Bool := FALSE;
      "SAFETY DOOR LOCK10.OUTPUT" : Bool := FALSE;
      SPARE_4 : Bool := FALSE;
      "SAFETY DOOR LOCK12.OUTPUT" : Bool := FALSE;
   END_VAR
BEGIN
END_DATA_BLOCK

